CASE ssMethodType OF
    SS_INITIALIZE: 
        temporalCounter_i1(timerAction := 1, maxTime := 0);
        temporalCounter_i2(timerAction := 1, maxTime := 0);
        temporalCounter_i1(timerAction := 1, maxTime := 0);
        is_active_c6_ChiefMaster := 0;
        is_c6_ChiefMaster := ChiefMaster_IN_NO_ACTIVE_CHILD_k;
        REQ_HV_ON := 0.0;
        ContactorState := 0.0;
    SS_OUTPUT: 
        (* Chart: '<S33>/Chart_REQ_HV_ON_Batt3' *)
        (* Gateway: ChiefMaster/Flow Logic/Battery HVControl/REQ_HV_ON_Batt/Chart_REQ_HV_ON_Batt3 *)
        (* During: ChiefMaster/Flow Logic/Battery HVControl/REQ_HV_ON_Batt/Chart_REQ_HV_ON_Batt3 *)

        IF is_active_c6_ChiefMaster = 0 THEN 
            (* Entry: ChiefMaster/Flow Logic/Battery HVControl/REQ_HV_ON_Batt/Chart_REQ_HV_ON_Batt3 *)
            is_active_c6_ChiefMaster := 1;
            (* Entry Internal: ChiefMaster/Flow Logic/Battery HVControl/REQ_HV_ON_Batt/Chart_REQ_HV_ON_Batt3 *)
            (* Transition: '<S42>:8' *)
            is_c6_ChiefMaster := ChiefMaster_IN_Default_f;
            (* Entry 'Default': '<S42>:7' *)
            (* '<S42>:7:2' REQ_HV_ON = 0 *)
            REQ_HV_ON := 0.0;
            (* '<S42>:7:3' ContactorState = 1 *)
            ContactorState := 1.0;
        ELSE 
            temp2 := FALSE;
            temp3 := FALSE;
            temp4 := FALSE;
            temp5 := FALSE;

            CASE is_c6_ChiefMaster OF
                ChiefMaster_IN_CONTACTOR_OFF_f: 
                    (* During 'CONTACTOR_OFF': '<S42>:18' *)
                    (* '<S42>:23:1' sf_internal_predicateOutput = InsulationReadyOK == false ||... *)
                    (* '<S42>:23:2' SDError_BB == true ||... *)
                    (* '<S42>:23:3' Software_Reset_KL15_BB == true ||... *)
                    (* '<S42>:23:4' KL15_CM_disable == true; *)

                    IF ((( NOT InsulationReadyOK) OR SDError_BB) OR (Software_Reset_KL15_BB = 1.0)) OR KL15_CM_disable THEN 
                        (* Transition: '<S42>:23' *)
                        is_c6_ChiefMaster := ChiefMaster_IN_Default_f;
                        (* Entry 'Default': '<S42>:7' *)
                        (* '<S42>:7:2' REQ_HV_ON = 0 *)
                        REQ_HV_ON := 0.0;
                        (* '<S42>:7:3' ContactorState = 1 *)
                        ContactorState := 1.0;
                    ELSE 
                        (* '<S42>:21:1' sf_internal_predicateOutput = after(2,sec) &&... *)
                        (* '<S42>:21:2' IMD_Active_BB1 == false &&... *)
                        (* '<S42>:21:3' IMD_Active_BB2 == false &&... *)
                        (* '<S42>:21:4' IMD_Active_BB3 == true &&... *)
                        (* '<S42>:21:5' MainHV_PlusMinus_Status == 0; *)
                        temporalCounter_i1(timerAction := 2, maxTime := 2000);

                        IF temporalCounter_i1.done THEN 

                            IF ((( NOT IMD_Active_BB1) AND ( NOT IMD_Active_BB2)) AND IMD_Active_BB3) AND ( NOT MainHV_PlusMinus_Status) THEN 
                                (* Transition: '<S42>:21' *)
                                temp3 := TRUE;
                            ELSE 
                                temp5 := TRUE;
                            END_IF;

                        ELSE 
                            temp5 := TRUE;
                        END_IF;

                    END_IF;

                ChiefMaster_IN_CONTACTOR_ON_b: 
                    (* During 'CONTACTOR_ON': '<S42>:20' *)
                    (* '<S42>:44:1' sf_internal_predicateOutput = (KL15_CM_disable == true || SDError_BB == true || System_SD == true) &&... *)
                    (* '<S42>:44:2' (MainHV_SD_OK == true || HV_REL_ON_BB3 == false); *)
                    tmp :=  NOT HV_REL_ON_BB3;

                    IF ((KL15_CM_disable OR SDError_BB) OR System_SD) AND (MainHV_SD_OK OR tmp) THEN 
                        (* Transition: '<S42>:44' *)
                        is_c6_ChiefMaster := ChiefMaster_IN_hold_k;
                        temporalCounter_i1(timerAction := 1, maxTime := 0);
                    ELSE 
                        (* '<S42>:51:1' sf_internal_predicateOutput = SDError_BB == true &&... *)
                        (* '<S42>:51:2' (HV_REL_ON_BB1 == true || HV_REL_ON_BB2 == true) &&... *)
                        (* '<S42>:51:3' (SafeToSD == true || HV_REL_ON_BB3 == false); *)
                        temp1 := HV_REL_ON_BB1 OR HV_REL_ON_BB2;

                        IF (SDError_BB AND temp1) AND (SafeToSD OR tmp) THEN 
                            (* Transition: '<S42>:51' *)
                            temp4 := TRUE;
                        ELSE 
                            (* '<S42>:66:1' sf_internal_predicateOutput = (HV_REL_ON_BB1 == true || HV_REL_ON_BB2 == true) &&... *)
                            (* '<S42>:66:2' REQ_HV_Open == true; *)

                            IF temp1 AND REQ_HV_Open THEN 
                                (* Transition: '<S42>:66' *)
                                temp4 := TRUE;
                            ELSE 
                                (* '<S42>:20:2' REQ_HV_ON = 1 *)
                                REQ_HV_ON := 1.0;
                                (* '<S42>:20:3' ContactorState = 3 *)
                                ContactorState := 3.0;
                            END_IF;

                        END_IF;

                    END_IF;

                ChiefMaster_IN_Default_f: 
                    (* During 'Default': '<S42>:7' *)
                    (* '<S42>:19:1' sf_internal_predicateOutput = IP_boChargeStop_Pressed == false &&... *)
                    (* '<S42>:19:2' KL15_CM_disable == false &&... *)
                    (* '<S42>:19:3' InsulationReadyOK == true &&... *)
                    (* '<S42>:19:4' SDError_BB == false &&... *)
                    (* '<S42>:19:5' System_SD == false; *)

                    IF (((( NOT IP_boChargeStop_Pressed) AND ( NOT KL15_CM_disable)) AND InsulationReadyOK) AND ( NOT SDError_BB)) AND ( NOT System_SD) THEN 
                        (* Transition: '<S42>:19' *)
                        is_c6_ChiefMaster := ChiefMaster_IN_CONTACTOR_OFF_f;
                        temporalCounter_i1(timerAction := 1, maxTime := 0);
                        temporalCounter_i2(timerAction := 1, maxTime := 0);
                        (* Entry 'CONTACTOR_OFF': '<S42>:18' *)
                        (* '<S42>:18:2' REQ_HV_ON = 0 *)
                        REQ_HV_ON := 0.0;
                        (* '<S42>:18:3' ContactorState = 2 *)
                        ContactorState := 2.0;
                    ELSE 
                        (* '<S42>:7:2' REQ_HV_ON = 0 *)
                        REQ_HV_ON := 0.0;
                        (* '<S42>:7:3' ContactorState = 1 *)
                        ContactorState := 1.0;
                    END_IF;

                ELSE
                    (* During 'hold': '<S42>:63' *)
                    (* '<S42>:64:1' sf_internal_predicateOutput = after(2,sec); *)
                    temporalCounter_i1(timerAction := 2, maxTime := 2000);

                    IF temporalCounter_i1.done THEN 
                        (* Transition: '<S42>:64' *)
                        is_c6_ChiefMaster := ChiefMaster_IN_Default_f;
                        (* Entry 'Default': '<S42>:7' *)
                        (* '<S42>:7:2' REQ_HV_ON = 0 *)
                        REQ_HV_ON := 0.0;
                        (* '<S42>:7:3' ContactorState = 1 *)
                        ContactorState := 1.0;
                    END_IF;

            END_CASE;


            IF temp5 THEN 
                (* '<S42>:28:1' sf_internal_predicateOutput = after(2,sec) &&... *)
                (* '<S42>:28:2' IMD_Active_BB3 == false &&... *)
                (* '<S42>:28:3' MainHV_PlusMinus_Status == 1 &&... *)
                (* '<S42>:28:4' (IMD_Active_BB1 == true || IMD_Active_BB2 ==true || IsolationMeasurementRequest == false) &&... *)
                (* '<S42>:28:5' SafeToCloseHV == true; *)
                temporalCounter_i2(timerAction := 2, maxTime := 2000);

                IF temporalCounter_i2.done THEN 

                    IF ((( NOT IMD_Active_BB3) AND MainHV_PlusMinus_Status) AND ((IMD_Active_BB1 OR IMD_Active_BB2) OR ( NOT IsolationMeasurementRequest))) AND SafeToCloseHV_n THEN 
                        (* Transition: '<S42>:28' *)
                        temp3 := TRUE;
                    ELSE 
                        temp2 := TRUE;
                    END_IF;

                ELSE 
                    temp2 := TRUE;
                END_IF;

            END_IF;


            IF temp4 THEN 
                is_c6_ChiefMaster := ChiefMaster_IN_Default_f;
                (* Entry 'Default': '<S42>:7' *)
                (* '<S42>:7:2' REQ_HV_ON = 0 *)
                REQ_HV_ON := 0.0;
                (* '<S42>:7:3' ContactorState = 1 *)
                ContactorState := 1.0;
            END_IF;


            IF temp3 THEN 
                is_c6_ChiefMaster := ChiefMaster_IN_CONTACTOR_ON_b;
                (* Entry 'CONTACTOR_ON': '<S42>:20' *)
                (* '<S42>:20:2' REQ_HV_ON = 1 *)
                REQ_HV_ON := 1.0;
                (* '<S42>:20:3' ContactorState = 3 *)
                ContactorState := 3.0;
            END_IF;


            IF temp2 THEN 
                (* '<S42>:18:2' REQ_HV_ON = 0 *)
                REQ_HV_ON := 0.0;
                (* '<S42>:18:3' ContactorState = 2 *)
                ContactorState := 2.0;
            END_IF;

        END_IF;

        (* End of Chart: '<S33>/Chart_REQ_HV_ON_Batt3' *)
END_CASE;

END_FUNCTION_BLOCK

// Device/Application/Chart_ContactorFB_State_Batt3
FUNCTION_BLOCK Chart_ContactorFB_State_Batt3
VAR_INPUT
	ssMethodType: SINT;
	HV_Minus_Sense_BB: BOOL;
	HV_Plus_Sense_BB: BOOL;
	REQ_HV_ON: LREAL;
END_VAR
VAR_OUTPUT
	Contactor_FB_State: LREAL;
END_VAR
VAR
	temporalCounter_i1: PLC_CODER_TIMER;
	is_c38_ChiefMaster: USINT;
	is_active_c38_ChiefMaster: USINT;
END_VAR



CASE ssMethodType OF
    SS_INITIALIZE: 
        temporalCounter_i1(timerAction := 1, maxTime := 0);
        is_active_c38_ChiefMaster := 0;
        is_c38_ChiefMaster := ChiefMaster_IN_NO_ACTIVE_CHILD_i;
        Contactor_FB_State := 0.0;
    SS_OUTPUT: 
        (* Chart: '<S33>/Chart_ContactorFB_State_Batt3' *)
        (* Gateway: ChiefMaster/Flow Logic/Battery HVControl/REQ_HV_ON_Batt/Chart_ContactorFB_State_Batt3 *)
        (* During: ChiefMaster/Flow Logic/Battery HVControl/REQ_HV_ON_Batt/Chart_ContactorFB_State_Batt3 *)

        IF is_active_c38_ChiefMaster = 0 THEN 
            (* Entry: ChiefMaster/Flow Logic/Battery HVControl/REQ_HV_ON_Batt/Chart_ContactorFB_State_Batt3 *)
            is_active_c38_ChiefMaster := 1;
            (* Entry Internal: ChiefMaster/Flow Logic/Battery HVControl/REQ_HV_ON_Batt/Chart_ContactorFB_State_Batt3 *)
            (* Transition: '<S39>:2' *)
            is_c38_ChiefMaster := ChiefMaster_IN_default_n;
            (* Entry 'default': '<S39>:1' *)
            (* '<S39>:1:2' Contactor_FB_State = 0 *)
            Contactor_FB_State := 0.0;
        ELSE 

            CASE is_c38_ChiefMaster OF
                ChiefMaster_IN_Error_c: 
                    (* During 'Error': '<S39>:12' *)
                    (* '<S39>:51:1' sf_internal_predicateOutput = REQ_HV_ON == 1; *)

                    IF REQ_HV_ON = 1.0 THEN 
                        (* Transition: '<S39>:51' *)
                        is_c38_ChiefMaster := ChiefMaster_IN_default_n;
                        (* Entry 'default': '<S39>:1' *)
                        (* '<S39>:1:2' Contactor_FB_State = 0 *)
                        Contactor_FB_State := 0.0;
                    ELSE 
                        (* '<S39>:12:2' Contactor_FB_State = 3 *)
                        Contactor_FB_State := 3.0;
                    END_IF;

                ChiefMaster_IN_Open_n: 
                    (* During 'Open': '<S39>:46' *)
                    (* '<S39>:50:1' sf_internal_predicateOutput = REQ_HV_ON == 1; *)

                    IF REQ_HV_ON = 1.0 THEN 
                        (* Transition: '<S39>:50' *)
                        is_c38_ChiefMaster := ChiefMaster_IN_default_n;
                        (* Entry 'default': '<S39>:1' *)
                        (* '<S39>:1:2' Contactor_FB_State = 0 *)
                        Contactor_FB_State := 0.0;
                    ELSE 
                        (* '<S39>:46:2' Contactor_FB_State = 1 *)
                        Contactor_FB_State := 1.0;
                    END_IF;

                ChiefMaster_IN_default_n: 
                    (* During 'default': '<S39>:1' *)
                    (* '<S39>:5:1' sf_internal_predicateOutput = REQ_HV_ON == 0; *)

                    IF REQ_HV_ON = 0.0 THEN 
                        (* Transition: '<S39>:5' *)
                        is_c38_ChiefMaster := ChiefMaster_IN_hold_h;
                        temporalCounter_i1(timerAction := 1, maxTime := 0);
                        (* Entry 'hold': '<S39>:4' *)
                        (* '<S39>:4:2' Contactor_FB_State = 0 *)
                        Contactor_FB_State := 0.0;
                    ELSE 
                        (* '<S39>:1:2' Contactor_FB_State = 0 *)
                        Contactor_FB_State := 0.0;
                    END_IF;

                ELSE
                    (* During 'hold': '<S39>:4' *)
                    (* '<S39>:13:1' sf_internal_predicateOutput = after(5,sec); *)
                    temporalCounter_i1(timerAction := 2, maxTime := 5000);

                    IF temporalCounter_i1.done THEN 
                        (* Transition: '<S39>:13' *)
                        is_c38_ChiefMaster := ChiefMaster_IN_Error_c;
                        (* Entry 'Error': '<S39>:12' *)
                        (* '<S39>:12:2' Contactor_FB_State = 3 *)
                        Contactor_FB_State := 3.0;
                    ELSE 
                        (* '<S39>:47:1' sf_internal_predicateOutput = HV_Plus_Sense_BB == false &&... *)
                        (* '<S39>:47:2' HV_Minus_Sense_BB == false; *)

                        IF ( NOT HV_Plus_Sense_BB) AND ( NOT HV_Minus_Sense_BB) THEN 
                            (* Transition: '<S39>:47' *)
                            is_c38_ChiefMaster := ChiefMaster_IN_Open_n;
                            (* Entry 'Open': '<S39>:46' *)
                            (* '<S39>:46:2' Contactor_FB_State = 1 *)
                            Contactor_FB_State := 1.0;
                        ELSE 
                            (* '<S39>:4:2' Contactor_FB_State = 0 *)
                            Contactor_FB_State := 0.0;
                        END_IF;

                    END_IF;

            END_CASE;

        END_IF;

        (* End of Chart: '<S33>/Chart_ContactorFB_State_Batt3' *)
END_CASE;

END_FUNCTION_BLOCK

// Device/Application/Chart_PrechargeStatus
FUNCTION_BLOCK Chart_PrechargeStatus
VAR_INPUT
	ssMethodType: SINT;
	REQ_MainHV_ON_Precharge: BOOL;
	LoadCurrent: BOOL;
	LoadVoltage: REAL;
	SystemVoltage: REAL;
	KL15_CM_diable: BOOL;
	MainHV_Minus_Status: LREAL;
END_VAR
VAR_OUTPUT
	Precharge_Satus: LREAL;
END_VAR
VAR
	temporalCounter_i2: PLC_CODER_TIMER;
	temporalCounter_i1: PLC_CODER_TIMER;
	is_c21_ChiefMaster: USINT;
	is_active_c21_ChiefMaster: USINT;
	temp1: BOOL;
END_VAR



CASE ssMethodType OF
    SS_INITIALIZE: 
        temporalCounter_i1(timerAction := 1, maxTime := 0);
        temporalCounter_i2(timerAction := 1, maxTime := 0);
        is_active_c21_ChiefMaster := 0;
        is_c21_ChiefMaster := ChiefMaster_IN_NO_ACTIVE_CHILD;
        Precharge_Satus := 0.0;
    SS_OUTPUT: 
        (* Chart: '<S13>/Chart_PrechargeStatus' *)
        (* Gateway: ChiefMaster/Flow Logic/BDU Control/BDUSystem/Chart_PrechargeStatus *)
        (* During: ChiefMaster/Flow Logic/BDU Control/BDUSystem/Chart_PrechargeStatus *)

        IF is_active_c21_ChiefMaster = 0 THEN 
            (* Entry: ChiefMaster/Flow Logic/BDU Control/BDUSystem/Chart_PrechargeStatus *)
            is_active_c21_ChiefMaster := 1;
            (* Entry Internal: ChiefMaster/Flow Logic/BDU Control/BDUSystem/Chart_PrechargeStatus *)
            (* Transition: '<S15>:4' *)
            is_c21_ChiefMaster := ChiefMaster_IN_Default;
            (* Entry 'Default': '<S15>:3' *)
            (* '<S15>:3:2' Precharge_Satus = 0 *)
            Precharge_Satus := 0.0;
        ELSE 

            CASE is_c21_ChiefMaster OF
                ChiefMaster_IN_Default: 
                    (* During 'Default': '<S15>:3' *)
                    (* '<S15>:20:1' sf_internal_predicateOutput = REQ_MainHV_ON_Precharge == true &&... *)
                    (* '<S15>:20:2' KL15_CM_diable == false; *)

                    IF REQ_MainHV_ON_Precharge AND ( NOT KL15_CM_diable) THEN 
                        (* Transition: '<S15>:20' *)
                        is_c21_ChiefMaster := ChiefMaster_IN_delay1;
                        temporalCounter_i1(timerAction := 1, maxTime := 0);
                        temporalCounter_i2(timerAction := 1, maxTime := 0);
                    ELSE 
                        (* '<S15>:3:2' Precharge_Satus = 0 *)
                        Precharge_Satus := 0.0;
                    END_IF;

                ChiefMaster_IN_PrechargeFail: 
                    (* During 'PrechargeFail': '<S15>:28' *)
                    (* Transition: '<S15>:37' *)
                    (* Transition: '<S15>:38' *)
                    (* '<S15>:35:1' sf_internal_predicateOutput = KL15_CM_diable == true; *)

                    IF KL15_CM_diable THEN 
                        (* Transition: '<S15>:35' *)
                        is_c21_ChiefMaster := ChiefMaster_IN_Default;
                        (* Entry 'Default': '<S15>:3' *)
                        (* '<S15>:3:2' Precharge_Satus = 0 *)
                        Precharge_Satus := 0.0;
                    ELSE 
                        (* '<S15>:28:2' Precharge_Satus = 2 *)
                        Precharge_Satus := 2.0;
                    END_IF;

                ChiefMaster_IN_PrechargeSuccess: 
                    (* During 'PrechargeSuccess': '<S15>:19' *)
                    (* Transition: '<S15>:32' *)
                    (* Transition: '<S15>:45' *)
                    (* '<S15>:46:1' sf_internal_predicateOutput = MainHV_Minus_Status == 1 ||... *)
                    (* '<S15>:46:2' MainHV_Minus_Status == 3; *)

                    IF (MainHV_Minus_Status = 1.0) OR (MainHV_Minus_Status = 3.0) THEN 
                        (* Transition: '<S15>:46' *)
                        is_c21_ChiefMaster := ChiefMaster_IN_Default;
                        (* Entry 'Default': '<S15>:3' *)
                        (* '<S15>:3:2' Precharge_Satus = 0 *)
                        Precharge_Satus := 0.0;
                    ELSE 
                        (* '<S15>:19:2' Precharge_Satus = 1 *)
                        Precharge_Satus := 1.0;
                    END_IF;

                ELSE
                    (* During 'delay1': '<S15>:26' *)
                    (* '<S15>:27:1' sf_internal_predicateOutput = after(500,msec) &&... *)
                    (* '<S15>:27:2' LoadCurrent == 0 &&... *)
                    (* '<S15>:27:3' abs(LoadVoltage - SystemVoltage) <= 5; *)
                    temp1 := FALSE;
                    temporalCounter_i2(timerAction := 2, maxTime := 500);

                    IF temporalCounter_i2.done THEN 

                        IF  NOT LoadCurrent THEN 

                            IF ABS(LoadVoltage - SystemVoltage) <= 5.0 THEN 
                                (* Transition: '<S15>:27' *)
                                is_c21_ChiefMaster := ChiefMaster_IN_PrechargeSuccess;
                                (* Entry 'PrechargeSuccess': '<S15>:19' *)
                                (* '<S15>:19:2' Precharge_Satus = 1 *)
                                Precharge_Satus := 1.0;
                            ELSE 
                                temp1 := TRUE;
                            END_IF;

                        ELSE 
                            temp1 := TRUE;
                        END_IF;

                    ELSE 
                        temp1 := TRUE;
                    END_IF;

                    temporalCounter_i1(timerAction := 2, maxTime := 3000);

                    IF temp1 AND temporalCounter_i1.done THEN 
                        (* '<S15>:25:1' sf_internal_predicateOutput = after(3,sec); *)
                        (* Transition: '<S15>:25' *)
                        is_c21_ChiefMaster := ChiefMaster_IN_PrechargeFail;
                        (* Entry 'PrechargeFail': '<S15>:28' *)
                        (* '<S15>:28:2' Precharge_Satus = 2 *)
                        Precharge_Satus := 2.0;
                    END_IF;

            END_CASE;

        END_IF;

        (* End of Chart: '<S13>/Chart_PrechargeStatus' *)
END_CASE;

END_FUNCTION_BLOCK

// Device/Application/Chart_SetDominantSwitch
FUNCTION_BLOCK Chart_SetDominantSwitch
VAR_INPUT
	ssMethodType: SINT;
	boData_In: BOOL;
	boReset: BOOL;
END_VAR
VAR_OUTPUT
	boData_Out: BOOL;
END_VAR
VAR
	is_active_c3_Library_DataProcessing_v1_1: USINT;
	is_c3_Library_DataProcessing_v1_1: USINT;
END_VAR



CASE ssMethodType OF
    SS_INITIALIZE: 
        is_active_c3_Library_DataProcessing_v1_1 := 0;
        is_c3_Library_DataProcessing_v1_1 := ChiefMaster_IN_NO_ACTIVE_CHILD_cn;
        boData_Out := FALSE;
    SS_OUTPUT: 
        (* Chart: '<S149>/Chart_SetDominantSwitch' *)
        (* Gateway: Lib_SetDominantSwitch/Chart_SetDominantSwitch *)
        (* During: Lib_SetDominantSwitch/Chart_SetDominantSwitch *)

        IF is_active_c3_Library_DataProcessing_v1_1 = 0 THEN 
            (* Entry: Lib_SetDominantSwitch/Chart_SetDominantSwitch *)
            is_active_c3_Library_DataProcessing_v1_1 := 1;
            (* Entry Internal: Lib_SetDominantSwitch/Chart_SetDominantSwitch *)
            (* Transition: '<S152>:10' *)
            is_c3_Library_DataProcessing_v1_1 := ChiefMaster_IN_Initial_state_g;
            (* Entry 'Initial_state': '<S152>:12' *)
            (* '<S152>:12:3' boData_Out = false; *)
            boData_Out := FALSE;
        ELSE 

            CASE is_c3_Library_DataProcessing_v1_1 OF
                ChiefMaster_IN_Initial_state_g: 
                    (* During 'Initial_state': '<S152>:12' *)
                    (* '<S152>:9:1' sf_internal_predicateOutput = boData_In == true; *)

                    IF boData_In THEN 
                        (* Transition: '<S152>:9' *)
                        is_c3_Library_DataProcessing_v1_1 := ChiefMaster_IN_state1_o;
                        (* Entry 'state1': '<S152>:6' *)
                        (* '<S152>:6:3' boData_Out = true; *)
                        boData_Out := TRUE;
                    ELSE 
                        (* '<S152>:12:3' boData_Out = false; *)
                        boData_Out := FALSE;
                    END_IF;

                ChiefMaster_IN_Reset_state_b: 
                    (* During 'Reset_state': '<S152>:4' *)
                    (* '<S152>:5:1' sf_internal_predicateOutput = boReset == false; *)

                    IF  NOT boReset THEN 
                        (* Transition: '<S152>:5' *)
                        is_c3_Library_DataProcessing_v1_1 := ChiefMaster_IN_Initial_state_g;
                        (* Entry 'Initial_state': '<S152>:12' *)
                        (* '<S152>:12:3' boData_Out = false; *)
                        boData_Out := FALSE;
                    ELSE 
                        (* '<S152>:4:3' boData_Out = false; *)
                        boData_Out := FALSE;
                    END_IF;

                ChiefMaster_IN_state1_o: 
                    (* During 'state1': '<S152>:6' *)
                    (* '<S152>:7:1' sf_internal_predicateOutput = boData_In == false; *)

                    IF  NOT boData_In THEN 
                        (* Transition: '<S152>:7' *)
                        is_c3_Library_DataProcessing_v1_1 := ChiefMaster_IN_state2_e;
                        (* Entry 'state2': '<S152>:8' *)
                        (* '<S152>:8:3' boData_Out = true; *)
                        boData_Out := TRUE;
                    ELSE 
                        (* '<S152>:6:3' boData_Out = true; *)
                        boData_Out := TRUE;
                    END_IF;

                ELSE
                    (* During 'state2': '<S152>:8' *)
                    (* '<S152>:11:1' sf_internal_predicateOutput = boReset == true; *)

                    IF boReset THEN 
                        (* Transition: '<S152>:11' *)
                        is_c3_Library_DataProcessing_v1_1 := ChiefMaster_IN_Reset_state_b;
                        (* Entry 'Reset_state': '<S152>:4' *)
                        (* '<S152>:4:3' boData_Out = false; *)
                        boData_Out := FALSE;
                    ELSE 
                        (* '<S152>:8:3' boData_Out = true; *)
                        boData_Out := TRUE;
                    END_IF;

            END_CASE;

        END_IF;

        (* End of Chart: '<S149>/Chart_SetDominantSwitch' *)
END_CASE;

END_FUNCTION_BLOCK

// Device/Application/EmergencySD
FUNCTION_BLOCK EmergencySD
VAR_INPUT
	ssMethodType: SINT;
	FL_boKL15_Reset: BOOL;
	IT_boEmergencySwitch_NC: BOOL;
	IT_boEmergencySwitch_NO: BOOL;
	IT_boHW_HVIL_BDU: BOOL;
	IT_boHW_HVIL_Components: BOOL;
	IT_boHW_HVIL_Battery: BOOL;
	IT_boHW_HVIL_Overrule: BOOL;
	IT_boHW_ResetButton_LED_NO_State: BOOL;
END_VAR
VAR_OUTPUT
	FL_boSS_System_ESD: BOOL;
	FL_u8SS_EmergencyStopState: USINT;
	FL_boHVIL_NOK: BOOL;
END_VAR
VAR
	is_active_c55_ChiefMaster: USINT;
	is_c55_ChiefMaster: USINT;
	temporalCounter_i1: PLC_CODER_TIMER;
	is_active_c28_ChiefMaster: USINT;
	is_c28_ChiefMaster: USINT;
	temporalCounter_i1_h: PLC_CODER_TIMER;
	i0_fcn_EmergencyButtonState: fcn_EmergencyButtonState;
	i0_HVIL_NOK: HVIL_NOK;
	rtb_out_j1: BOOL;
	rtb_out_h: BOOL;
	rtb_TmpSignalConversionAtfcn_EmergencyButtonStateInport2: BOOL;
END_VAR



CASE ssMethodType OF
    SS_INITIALIZE: 
        (* SystemInitialize for Chart: '<S140>/EmergencySwitch_Input_Delay1' *)
        temporalCounter_i1(timerAction := 1, maxTime := 0);
        is_active_c55_ChiefMaster := 0;
        is_c55_ChiefMaster := ChiefMaster_IN_NO_ACTIVE_CHILD_l;
        (* SystemInitialize for Chart: '<S140>/EmergencySwitch_Input_Delay' *)
        temporalCounter_i1_h(timerAction := 1, maxTime := 0);
        is_active_c28_ChiefMaster := 0;
        is_c28_ChiefMaster := ChiefMaster_IN_NO_ACTIVE_CHILD_l;
        (* SystemInitialize for Chart: '<S140>/EmergencySwitch_Input_Delay1' incorporates:
         *  Chart: '<S140>/EmergencySwitch_Input_Delay' *)
        i0_fcn_EmergencyButtonState(ssMethodType := SS_INITIALIZE, IP_boVS_EmergencySwitch_NO_S1 := FALSE, IP_boVS_EmergencySwitch_NC_S2 := rtb_TmpSignalConversionAtfcn_EmergencyButtonStateInport2, IP_boVS_EmergencySwitch_NC_S3 := FALSE, b_reset := rtb_TmpSignalConversionAtfcn_EmergencyButtonStateInport2);
        FL_u8SS_EmergencyStopState := i0_fcn_EmergencyButtonState.FL_u8VS_EmergencyStopState;
        i0_HVIL_NOK(ssMethodType := SS_INITIALIZE, boReset := rtb_TmpSignalConversionAtfcn_EmergencyButtonStateInport2, IT_boHW_HVIL_BDU := IT_boHW_HVIL_BDU, IT_boHW_HVIL_Components := IT_boHW_HVIL_Components, IT_boHW_HVIL_Battery := IT_boHW_HVIL_Battery);
    SS_OUTPUT: 
        (* Logic: '<S112>/AND' incorporates:
         *  Logic: '<S112>/NOT' *)
        rtb_TmpSignalConversionAtfcn_EmergencyButtonStateInport2 := IT_boHW_ResetButton_LED_NO_State AND ( NOT FL_boKL15_Reset);
        (* Chart: '<S140>/EmergencySwitch_Input_Delay1' *)
        (* Gateway: ChiefMaster/Flow Logic/System Status/EmergencySD/Emergency_Switch_Control/EmergencySwitch_Input_Delay1 *)
        (* During: ChiefMaster/Flow Logic/System Status/EmergencySD/Emergency_Switch_Control/EmergencySwitch_Input_Delay1 *)

        IF is_active_c55_ChiefMaster = 0 THEN 
            (* Entry: ChiefMaster/Flow Logic/System Status/EmergencySD/Emergency_Switch_Control/EmergencySwitch_Input_Delay1 *)
            is_active_c55_ChiefMaster := 1;
            (* Entry Internal: ChiefMaster/Flow Logic/System Status/EmergencySD/Emergency_Switch_Control/EmergencySwitch_Input_Delay1 *)
            (* Transition: '<S143>:2' *)
            is_c55_ChiefMaster := ChiefMaster_IN_Initial;
            (* Entry 'Initial': '<S143>:1' *)
            (* '<S143>:1:3' out = IP_boVS_EmergensySwitch; *)
            rtb_out_j1 := IT_boEmergencySwitch_NO;
        ELSE 

            CASE is_c55_ChiefMaster OF
                ChiefMaster_IN_After_delay: 
                    (* During 'After_delay': '<S143>:4' *)
                    (* '<S143>:10:1' sf_internal_predicateOutput = IP_boVS_EmergensySwitch == true; *)

                    IF IT_boEmergencySwitch_NO THEN 
                        (* Transition: '<S143>:10' *)
                        is_c55_ChiefMaster := ChiefMaster_IN_Initial;
                        (* Entry 'Initial': '<S143>:1' *)
                        (* '<S143>:1:3' out = IP_boVS_EmergensySwitch; *)
                        rtb_out_j1 := TRUE;
                    ELSE 
                        (* '<S143>:4:3' out = IP_boVS_EmergensySwitch; *)
                        rtb_out_j1 := FALSE;
                    END_IF;

                ChiefMaster_IN_Delay_a: 
                    (* During 'Delay': '<S143>:3' *)
                    (* '<S143>:6:1' sf_internal_predicateOutput = after(10, msec); *)
                    temporalCounter_i1(timerAction := 2, maxTime := 10);

                    IF temporalCounter_i1.done THEN 
                        (* Transition: '<S143>:6' *)
                        is_c55_ChiefMaster := ChiefMaster_IN_After_delay;
                        (* Entry 'After_delay': '<S143>:4' *)
                        (* '<S143>:4:3' out = IP_boVS_EmergensySwitch; *)
                        rtb_out_j1 := IT_boEmergencySwitch_NO;
                    ELSE 
                        (* '<S143>:3:3' out = false; *)
                        rtb_out_j1 := FALSE;
                    END_IF;

                ELSE
                    (* During 'Initial': '<S143>:1' *)
                    (* '<S143>:5:1' sf_internal_predicateOutput = IP_boVS_EmergensySwitch == false; *)

                    IF  NOT IT_boEmergencySwitch_NO THEN 
                        (* Transition: '<S143>:5' *)
                        is_c55_ChiefMaster := ChiefMaster_IN_Delay_a;
                        temporalCounter_i1(timerAction := 1, maxTime := 0);
                        (* Entry 'Delay': '<S143>:3' *)
                        (* '<S143>:3:3' out = false; *)
                        rtb_out_j1 := FALSE;
                    ELSE 
                        (* '<S143>:1:3' out = IP_boVS_EmergensySwitch; *)
                        rtb_out_j1 := TRUE;
                    END_IF;

            END_CASE;

        END_IF;

        (* End of Chart: '<S140>/EmergencySwitch_Input_Delay1' *)
        

        (* Chart: '<S140>/EmergencySwitch_Input_Delay' *)
        (* Gateway: ChiefMaster/Flow Logic/System Status/EmergencySD/Emergency_Switch_Control/EmergencySwitch_Input_Delay *)
        (* During: ChiefMaster/Flow Logic/System Status/EmergencySD/Emergency_Switch_Control/EmergencySwitch_Input_Delay *)

        IF is_active_c28_ChiefMaster = 0 THEN 
            (* Entry: ChiefMaster/Flow Logic/System Status/EmergencySD/Emergency_Switch_Control/EmergencySwitch_Input_Delay *)
            is_active_c28_ChiefMaster := 1;
            (* Entry Internal: ChiefMaster/Flow Logic/System Status/EmergencySD/Emergency_Switch_Control/EmergencySwitch_Input_Delay *)
            (* Transition: '<S142>:2' *)
            is_c28_ChiefMaster := ChiefMaster_IN_Initial;
            (* Entry 'Initial': '<S142>:1' *)
            (* '<S142>:1:3' out = IP_boVS_EmergensySwitch; *)
            rtb_out_h := IT_boEmergencySwitch_NC;
        ELSE 

            CASE is_c28_ChiefMaster OF
                ChiefMaster_IN_After_delay: 
                    (* During 'After_delay': '<S142>:4' *)
                    (* '<S142>:10:1' sf_internal_predicateOutput = IP_boVS_EmergensySwitch == true; *)

                    IF IT_boEmergencySwitch_NC THEN 
                        (* Transition: '<S142>:10' *)
                        is_c28_ChiefMaster := ChiefMaster_IN_Initial;
                        (* Entry 'Initial': '<S142>:1' *)
                        (* '<S142>:1:3' out = IP_boVS_EmergensySwitch; *)
                        rtb_out_h := TRUE;
                    ELSE 
                        (* '<S142>:4:3' out = IP_boVS_EmergensySwitch; *)
                        rtb_out_h := FALSE;
                    END_IF;

                ChiefMaster_IN_Delay_a: 
                    (* During 'Delay': '<S142>:3' *)
                    (* '<S142>:6:1' sf_internal_predicateOutput = after(10, msec); *)
                    temporalCounter_i1_h(timerAction := 2, maxTime := 10);

                    IF temporalCounter_i1_h.done THEN 
                        (* Transition: '<S142>:6' *)
                        is_c28_ChiefMaster := ChiefMaster_IN_After_delay;
                        (* Entry 'After_delay': '<S142>:4' *)
                        (* '<S142>:4:3' out = IP_boVS_EmergensySwitch; *)
                        rtb_out_h := IT_boEmergencySwitch_NC;
                    ELSE 
                        (* '<S142>:3:3' out = true; *)
                        rtb_out_h := TRUE;
                    END_IF;

                ELSE
                    (* During 'Initial': '<S142>:1' *)
                    (* '<S142>:5:1' sf_internal_predicateOutput = IP_boVS_EmergensySwitch == false; *)

                    IF  NOT IT_boEmergencySwitch_NC THEN 
                        (* Transition: '<S142>:5' *)
                        is_c28_ChiefMaster := ChiefMaster_IN_Delay_a;
                        temporalCounter_i1_h(timerAction := 1, maxTime := 0);
                        (* Entry 'Delay': '<S142>:3' *)
                        (* '<S142>:3:3' out = true; *)
                        rtb_out_h := TRUE;
                    ELSE 
                        (* '<S142>:1:3' out = IP_boVS_EmergensySwitch; *)
                        rtb_out_h := TRUE;
                    END_IF;

            END_CASE;

        END_IF;

        (* End of Chart: '<S140>/EmergencySwitch_Input_Delay' *)
        

        (* SignalConversion: '<S140>/TmpSignal ConversionAtfcn_EmergencyButtonStateInport2' *)
        i0_fcn_EmergencyButtonState(ssMethodType := SS_OUTPUT, IP_boVS_EmergencySwitch_NO_S1 := rtb_out_j1, IP_boVS_EmergencySwitch_NC_S2 := rtb_out_h, IP_boVS_EmergencySwitch_NC_S3 := rtb_out_h, b_reset := rtb_TmpSignalConversionAtfcn_EmergencyButtonStateInport2);
        FL_u8SS_EmergencyStopState := i0_fcn_EmergencyButtonState.FL_u8VS_EmergencyStopState;
        i0_HVIL_NOK(ssMethodType := SS_OUTPUT, boReset := rtb_TmpSignalConversionAtfcn_EmergencyButtonStateInport2, IT_boHW_HVIL_BDU := IT_boHW_HVIL_BDU, IT_boHW_HVIL_Components := IT_boHW_HVIL_Components, IT_boHW_HVIL_Battery := IT_boHW_HVIL_Battery);
        FL_boSS_System_ESD := i0_HVIL_NOK.FL_boSS_HVIL_NOK;
        (* Switch: '<S112>/Switch' incorporates:
         *  Constant: '<S112>/Constant' *)

        IF IT_boHW_HVIL_Overrule THEN 
            FL_boHVIL_NOK := FALSE;
        ELSE 
            FL_boHVIL_NOK := FL_boSS_System_ESD;
        END_IF;

        (* End of Switch: '<S112>/Switch' *)
        

        (* Logic: '<S112>/OR1' incorporates:
         *  Constant: '<S139>/Constant'
         *  RelationalOperator: '<S139>/Compare' *)
        FL_boSS_System_ESD := (FL_u8SS_EmergencyStopState >= 1) OR FL_boHVIL_NOK;
END_CASE;

END_FUNCTION_BLOCK

// Device/Application/fcn_EmergencyButtonState
FUNCTION_BLOCK fcn_EmergencyButtonState
VAR_INPUT
	ssMethodType: SINT;
	IP_boVS_EmergencySwitch_NO_S1: BOOL;
	IP_boVS_EmergencySwitch_NC_S2: BOOL;
	IP_boVS_EmergencySwitch_NC_S3: BOOL;
	b_reset: BOOL;
END_VAR
VAR_OUTPUT
	FL_u8VS_EmergencyStopState: USINT;
END_VAR
VAR
	is_active_c29_ChiefMaster: USINT;
	is_c29_ChiefMaster: USINT;
	In_prv: USINT;
END_VAR



CASE ssMethodType OF
    SS_INITIALIZE: 
        (* SystemInitialize for Chart: '<S144>/Chart' *)
        is_active_c29_ChiefMaster := 0;
        is_c29_ChiefMaster := ChiefMaster_IN_NO_ACTIVE_CHILD_b;
        In_prv := 0;
        FL_u8VS_EmergencyStopState := 0;
    SS_OUTPUT: 
        (* Switch: '<S144>/Switch1' incorporates:
         *  Constant: '<S144>/NotPressed'
         *  Logic: '<S144>/AND1'
         *  Logic: '<S144>/AND3'
         *  Logic: '<S144>/AND4'
         *  Logic: '<S144>/AND5'
         *  Switch: '<S144>/Switch' *)

        IF ( NOT IP_boVS_EmergencySwitch_NO_S1) AND (IP_boVS_EmergencySwitch_NC_S2 AND IP_boVS_EmergencySwitch_NC_S3) THEN 
            FL_u8VS_EmergencyStopState := 0;
        ELSIF IP_boVS_EmergencySwitch_NO_S1 AND (( NOT IP_boVS_EmergencySwitch_NC_S2) AND ( NOT IP_boVS_EmergencySwitch_NC_S3)) THEN 
            (* Switch: '<S144>/Switch' incorporates:
             *  Constant: '<S144>/Pressed' *)
            FL_u8VS_EmergencyStopState := 1;
        ELSE 
            (* Switch: '<S144>/Switch' incorporates:
             *  Constant: '<S144>/Error' *)
            FL_u8VS_EmergencyStopState := 2;
        END_IF;

        (* End of Switch: '<S144>/Switch1' *)
        

        (* Chart: '<S144>/Chart' *)
        (* Gateway: ChiefMaster/Flow Logic/System Status/EmergencySD/Emergency_Switch_Control/fcn_EmergencyButtonState/Chart *)
        (* During: ChiefMaster/Flow Logic/System Status/EmergencySD/Emergency_Switch_Control/fcn_EmergencyButtonState/Chart *)

        IF is_active_c29_ChiefMaster = 0 THEN 
            (* Entry: ChiefMaster/Flow Logic/System Status/EmergencySD/Emergency_Switch_Control/fcn_EmergencyButtonState/Chart *)
            is_active_c29_ChiefMaster := 1;
            (* Entry Internal: ChiefMaster/Flow Logic/System Status/EmergencySD/Emergency_Switch_Control/fcn_EmergencyButtonState/Chart *)
            (* Transition: '<S145>:5' *)
            is_c29_ChiefMaster := ChiefMaster_IN_Initial_state;
            (* Entry 'Initial_state': '<S145>:7' *)
            (* '<S145>:7:3' Out = In; *)
        ELSE 

            CASE is_c29_ChiefMaster OF
                ChiefMaster_IN_Initial_state: 
                    (* During 'Initial_state': '<S145>:7' *)
                    (* '<S145>:9:1' sf_internal_predicateOutput = In > uint8(0); *)

                    IF FL_u8VS_EmergencyStopState > 0 THEN 
                        (* Transition: '<S145>:9' *)
                        is_c29_ChiefMaster := ChiefMaster_IN_state1;
                        (* Entry 'state1': '<S145>:2' *)
                        (* '<S145>:2:3' Out = In; *)
                        (* '<S145>:2:4' In_prv = In; *)
                        In_prv := FL_u8VS_EmergencyStopState;
                    END_IF;

                ChiefMaster_IN_Reset_state: 
                    (* During 'Reset_state': '<S145>:1' *)
                    (* '<S145>:8:1' sf_internal_predicateOutput = reset == false; *)

                    IF  NOT b_reset THEN 
                        (* Transition: '<S145>:8' *)
                        is_c29_ChiefMaster := ChiefMaster_IN_Initial_state;
                        (* Entry 'Initial_state': '<S145>:7' *)
                        (* '<S145>:7:3' Out = In; *)
                    ELSE 
                        (* '<S145>:1:3' Out = uint8(0); *)
                        FL_u8VS_EmergencyStopState := 0;
                    END_IF;

                ChiefMaster_IN_state1: 
                    (* During 'state1': '<S145>:2' *)
                    (* '<S145>:6:1' sf_internal_predicateOutput = In == uint8(0); *)

                    IF FL_u8VS_EmergencyStopState = 0 THEN 
                        (* Transition: '<S145>:6' *)
                        is_c29_ChiefMaster := ChiefMaster_IN_state2;
                        (* Entry 'state2': '<S145>:3' *)
                        (* '<S145>:3:3' Out = In_prv; *)
                        FL_u8VS_EmergencyStopState := In_prv;
                    ELSE 
                        (* '<S145>:2:3' Out = In; *)
                        (* '<S145>:2:4' In_prv = In; *)
                        In_prv := FL_u8VS_EmergencyStopState;
                    END_IF;

                ELSE
                    (* During 'state2': '<S145>:3' *)
                    (* '<S145>:4:1' sf_internal_predicateOutput = reset == true; *)

                    IF b_reset THEN 
                        (* Transition: '<S145>:4' *)
                        is_c29_ChiefMaster := ChiefMaster_IN_Reset_state;
                        (* Entry 'Reset_state': '<S145>:1' *)
                        (* '<S145>:1:3' Out = uint8(0); *)
                        FL_u8VS_EmergencyStopState := 0;
                    ELSE 
                        (* '<S145>:3:3' Out = In_prv; *)
                        FL_u8VS_EmergencyStopState := In_prv;
                    END_IF;

            END_CASE;

        END_IF;

        (* End of Chart: '<S144>/Chart' *)
END_CASE;

END_FUNCTION_BLOCK

// Device/Application/HVIL_NOK
FUNCTION_BLOCK HVIL_NOK
VAR_INPUT
	ssMethodType: SINT;
	boReset: BOOL;
	IT_boHW_HVIL_BDU: BOOL;
	IT_boHW_HVIL_Components: BOOL;
	IT_boHW_HVIL_Battery: BOOL;
END_VAR
VAR_OUTPUT
	FL_boSS_HVIL_NOK: BOOL;
END_VAR
VAR
	i0_Chart_SetDominantSwitch: Chart_SetDominantSwitch;
	i1_Chart_SetDominantSwitch: Chart_SetDominantSwitch;
	i2_Chart_SetDominantSwitch: Chart_SetDominantSwitch;
	rtb_Compare_jkc: BOOL;
	rtb_boData_Out_f5: BOOL;
	rtb_Compare_h3: BOOL;
	rtb_Compare_n45: BOOL;
END_VAR



CASE ssMethodType OF
    SS_INITIALIZE: 
        i0_Chart_SetDominantSwitch(ssMethodType := SS_INITIALIZE, boData_In := rtb_Compare_jkc, boReset := boReset);
        rtb_boData_Out_f5 := i0_Chart_SetDominantSwitch.boData_Out;
        i1_Chart_SetDominantSwitch(ssMethodType := SS_INITIALIZE, boData_In := rtb_Compare_h3, boReset := boReset);
        rtb_Compare_jkc := i1_Chart_SetDominantSwitch.boData_Out;
        i2_Chart_SetDominantSwitch(ssMethodType := SS_INITIALIZE, boData_In := rtb_Compare_n45, boReset := boReset);
        rtb_Compare_h3 := i2_Chart_SetDominantSwitch.boData_Out;
    SS_OUTPUT: 
        (* RelationalOperator: '<S146>/Compare' *)
        i0_Chart_SetDominantSwitch(ssMethodType := SS_OUTPUT, boData_In :=  NOT IT_boHW_HVIL_BDU, boReset := boReset);
        rtb_boData_Out_f5 := i0_Chart_SetDominantSwitch.boData_Out;
        (* RelationalOperator: '<S147>/Compare' *)
        i1_Chart_SetDominantSwitch(ssMethodType := SS_OUTPUT, boData_In :=  NOT IT_boHW_HVIL_Components, boReset := boReset);
        rtb_Compare_jkc := i1_Chart_SetDominantSwitch.boData_Out;
        (* RelationalOperator: '<S148>/Compare' *)
        i2_Chart_SetDominantSwitch(ssMethodType := SS_OUTPUT, boData_In :=  NOT IT_boHW_HVIL_Battery, boReset := boReset);
        rtb_Compare_h3 := i2_Chart_SetDominantSwitch.boData_Out;
        (* Logic: '<S141>/OR' *)
        FL_boSS_HVIL_NOK := (rtb_boData_Out_f5 OR rtb_Compare_jkc) OR rtb_Compare_h3;
END_CASE;

END_FUNCTION_BLOCK

// Device/Application/Input_Delay
FUNCTION_BLOCK Input_Delay
VAR_INPUT
	ssMethodType: SINT;
	IP_u8HW_IN_delay_ms_m: UINT;
	Input: BOOL;
END_VAR
VAR_OUTPUT
	out: BOOL;
END_VAR
VAR
	is_active_c2_ChiefMaster: USINT;
	is_c2_ChiefMaster: USINT;
	temporalCounter_i1: PLC_CODER_TIMER;
END_VAR



CASE ssMethodType OF
    SS_INITIALIZE: 
        temporalCounter_i1(timerAction := 1, maxTime := 0);
        is_active_c2_ChiefMaster := 0;
        is_c2_ChiefMaster := ChiefMaster_IN_NO_ACTIVE_CHILD_an;
        out := FALSE;
    SS_OUTPUT: 
        (* Chart: '<S392>/Input_Delay' *)
        (* Gateway: ChiefMaster/Input Processing/HW Inputs/Subsystem/Input_Delay *)
        (* During: ChiefMaster/Input Processing/HW Inputs/Subsystem/Input_Delay *)

        IF is_active_c2_ChiefMaster = 0 THEN 
            (* Entry: ChiefMaster/Input Processing/HW Inputs/Subsystem/Input_Delay *)
            is_active_c2_ChiefMaster := 1;
            (* Entry Internal: ChiefMaster/Input Processing/HW Inputs/Subsystem/Input_Delay *)
            (* Transition: '<S418>:2' *)
            is_c2_ChiefMaster := ChiefMaster_IN_Initial_k;
            temporalCounter_i1(timerAction := 1, maxTime := 0);
            (* Entry 'Initial': '<S418>:1' *)
            (* '<S418>:1:3' out = true; *)
            out := TRUE;
        ELSE 

            CASE is_c2_ChiefMaster OF
                ChiefMaster_IN_After_delay_p: 
                    (* During 'After_delay': '<S418>:4' *)
                    (* '<S418>:4:3' out = Input; *)
                    out := Input;
                ELSE
                    (* During 'Initial': '<S418>:1' *)
                    (* '<S418>:6:1' sf_internal_predicateOutput = after(IP_u8HW_IN_delay_ms, msec); *)
                    temporalCounter_i1(timerAction := 2, maxTime := UINT_TO_DINT(IP_u8HW_IN_delay_ms_m));

                    IF temporalCounter_i1.done THEN 
                        (* Transition: '<S418>:6' *)
                        is_c2_ChiefMaster := ChiefMaster_IN_After_delay_p;
                        (* Entry 'After_delay': '<S418>:4' *)
                        (* '<S418>:4:3' out = Input; *)
                        out := Input;
                    ELSE 
                        (* '<S418>:1:3' out = true; *)
                        out := TRUE;
                    END_IF;

            END_CASE;

        END_IF;

        (* End of Chart: '<S392>/Input_Delay' *)
END_CASE;

END_FUNCTION_BLOCK

// Device/Application/SDError
FUNCTION_BLOCK SDError
VAR_INPUT
	ssMethodType: SINT;
	FL_boKL15_Reset: BOOL;
	IT_Databus: USINT;
	IT_Databus_m: BOOL;
	IT_Databus_n: BOOL;
	IT_Databus_a: BOOL;
	IT_Databus_o: BOOL;
	IT_Databus_or: BOOL;
	IT_Databus_i: BOOL;
	IT_Databus_c: REAL;
	IT_Databus_o3: REAL;
	IT_Databus_e: REAL;
	IT_Databus_n0: BOOL;
	IT_Databus_ep: BOOL;
	IT_Databus_l: BOOL;
	IT_Databus_f: BOOL;
	IT_Databus_k: BOOL;
	IT_Databus_g: BOOL;
	IT_Databus_b: BOOL;
	IT_Databus_d: BOOL;
	IT_Databus_h: BOOL;
	IT_Databus_j: BOOL;
	IT_Databus_ja: BOOL;
	IT_Databus_if: BOOL;
	FL_BDUControl_Databus: LREAL;
	FL_BDUControl_Databus_o: LREAL;
	FL_BDUControl_Databus_n: LREAL;
	FL_BatteryBox_HVControl_Databus: LREAL;
	FL_BatteryBox_HVControl_Databus_b: LREAL;
	FL_BatteryBox_HVControl_Databus_a: LREAL;
	FL_u8SS_EmergencySD: BOOL;
END_VAR
VAR_OUTPUT
	FL_boSS_System_SD: BOOL;
	FL_u8SS_System_SD_ErrorCode: USINT;
END_VAR
VAR
	is_active_c39_ChiefMaster: USINT;
	is_c39_ChiefMaster: USINT;
	DelayInput1_DSTATE: LREAL;
	DelayInput1_DSTATE_a: LREAL;
	DelayInput1_DSTATE_j: LREAL;
	i0_BDU_Error: BDU_Error;
	i0_Chart_ek: Chart_ek;
	i1_Chart_ek: Chart_ek;
	i2_Chart_ek: Chart_ek;
	i0_IMD_SD: IMD_SD;
	rtb_OR1_c: BOOL;
	rtb_Switch_k: BOOL;
	rtb_FixPtRelationalOperator_h5: BOOL;
	rtb_Out_nh: BOOL;
	rtb_FixPtRelationalOperator_m: BOOL;
	rtb_Out_lz: BOOL;
	rtb_Switch1_j1g: BOOL;
	rtb_Compare_jn: BOOL;
	temp1: DINT;
END_VAR



CASE ssMethodType OF
    SS_INITIALIZE: 
        (* InitializeConditions for UnitDelay: '<S181>/Delay Input1'
         *
         * Block description for '<S181>/Delay Input1':
         *  
         *  Store in Global RAM *)
        DelayInput1_DSTATE := 0.0;
        (* InitializeConditions for UnitDelay: '<S182>/Delay Input1'
         *
         * Block description for '<S182>/Delay Input1':
         *  
         *  Store in Global RAM *)
        DelayInput1_DSTATE_a := 0.0;
        (* InitializeConditions for UnitDelay: '<S183>/Delay Input1'
         *
         * Block description for '<S183>/Delay Input1':
         *  
         *  Store in Global RAM *)
        DelayInput1_DSTATE_j := 0.0;
        i0_BDU_Error(ssMethodType := SS_INITIALIZE, Main_REL_Databus := FL_BDUControl_Databus, Main_REL_Databus_c := FL_BDUControl_Databus_o, Main_REL_Databus_p := FL_BDUControl_Databus_n);
        i0_Chart_ek(ssMethodType := SS_INITIALIZE, In := rtb_FixPtRelationalOperator_h5, REQ_HV_ON_BB := rtb_FixPtRelationalOperator_h5, KL15_CM_Reset := FL_boKL15_Reset);
        rtb_Out_nh := i0_Chart_ek.Out;
        i1_Chart_ek(ssMethodType := SS_INITIALIZE, In := rtb_FixPtRelationalOperator_m, REQ_HV_ON_BB := rtb_FixPtRelationalOperator_m, KL15_CM_Reset := FL_boKL15_Reset);
        rtb_FixPtRelationalOperator_h5 := i1_Chart_ek.Out;
        i2_Chart_ek(ssMethodType := SS_INITIALIZE, In := rtb_FixPtRelationalOperator_m, REQ_HV_ON_BB := rtb_FixPtRelationalOperator_m, KL15_CM_Reset := FL_boKL15_Reset);
        rtb_Out_lz := i2_Chart_ek.Out;
        i0_IMD_SD(ssMethodType := SS_INITIALIZE, BatteryPackSignals := IT_Databus_f, BatteryPackSignals_g := IT_Databus_m, BatteryPackSignals_f := IT_Databus_k, BatteryPackSignals_d := IT_Databus_a, BatteryPackSignals_c := IT_Databus_g, BatteryPackSignals_c4 := IT_Databus_or, BatteryPackSignals_dh := IT_Databus_b, BatteryPackSignals_k := IT_Databus_d, BatteryPackSignals_g5 := IT_Databus_h, BatteryPackSignals_b := IT_Databus_j, BatteryPackSignals_di := IT_Databus_ja, BatteryPackSignals_n := IT_Databus_if);
        (* SystemInitialize for Chart: '<S115>/Chart' *)
        is_active_c39_ChiefMaster := 0;
        is_c39_ChiefMaster := ChiefMaster_IN_NO_ACTIVE_CHILD_cs;
        FL_boSS_System_SD := FALSE;
    SS_OUTPUT: 
        (* RelationalOperator: '<S158>/Compare' incorporates:
         *  Constant: '<S158>/Constant' *)
        rtb_FixPtRelationalOperator_m := IT_Databus = 0;
        (* Switch: '<S164>/Switch' incorporates:
         *  Constant: '<S164>/Constant'
         *  Logic: '<S164>/AND' *)

        IF IT_Databus_m AND rtb_FixPtRelationalOperator_m THEN 
            rtb_Switch_k := IT_Databus_n;
        ELSE 
            rtb_Switch_k := FALSE;
        END_IF;

        (* End of Switch: '<S164>/Switch' *)
        

        (* Switch: '<S163>/Switch1' incorporates:
         *  Constant: '<S163>/Constant'
         *  Logic: '<S163>/AND1' *)

        IF IT_Databus_a AND rtb_FixPtRelationalOperator_m THEN 
            rtb_Switch1_j1g := IT_Databus_o;
        ELSE 
            rtb_Switch1_j1g := FALSE;
        END_IF;

        (* End of Switch: '<S163>/Switch1' *)
        

        (* Switch: '<S162>/Switch2' incorporates:
         *  Constant: '<S162>/Constant'
         *  Logic: '<S162>/AND2' *)

        IF IT_Databus_or AND rtb_FixPtRelationalOperator_m THEN 
            rtb_FixPtRelationalOperator_m := IT_Databus_i;
        ELSE 
            rtb_FixPtRelationalOperator_m := FALSE;
        END_IF;

        (* End of Switch: '<S162>/Switch2' *)
        i0_BDU_Error(ssMethodType := SS_OUTPUT, Main_REL_Databus := FL_BDUControl_Databus, Main_REL_Databus_c := FL_BDUControl_Databus_o, Main_REL_Databus_p := FL_BDUControl_Databus_n);
        rtb_OR1_c := i0_BDU_Error.BDU_Error_lg;
        (* RelationalOperator: '<S181>/FixPt Relational Operator' incorporates:
         *  Constant: '<S176>/Constant'
         *  RelationalOperator: '<S176>/Compare'
         *  UnitDelay: '<S181>/Delay Input1'
         *
         * Block description for '<S181>/Delay Input1':
         *  
         *  Store in Global RAM *)
        i0_Chart_ek(ssMethodType := SS_OUTPUT, In := FL_BatteryBox_HVControl_Databus < DelayInput1_DSTATE, REQ_HV_ON_BB := FL_BatteryBox_HVControl_Databus = 0.0, KL15_CM_Reset := FL_boKL15_Reset);
        rtb_Out_nh := i0_Chart_ek.Out;
        (* RelationalOperator: '<S182>/FixPt Relational Operator' incorporates:
         *  Constant: '<S178>/Constant'
         *  RelationalOperator: '<S178>/Compare'
         *  UnitDelay: '<S182>/Delay Input1'
         *
         * Block description for '<S182>/Delay Input1':
         *  
         *  Store in Global RAM *)
        i1_Chart_ek(ssMethodType := SS_OUTPUT, In := FL_BatteryBox_HVControl_Databus_b < DelayInput1_DSTATE_a, REQ_HV_ON_BB := FL_BatteryBox_HVControl_Databus_b = 0.0, KL15_CM_Reset := FL_boKL15_Reset);
        rtb_FixPtRelationalOperator_h5 := i1_Chart_ek.Out;
        (* RelationalOperator: '<S183>/FixPt Relational Operator' incorporates:
         *  Constant: '<S180>/Constant'
         *  RelationalOperator: '<S180>/Compare'
         *  UnitDelay: '<S183>/Delay Input1'
         *
         * Block description for '<S183>/Delay Input1':
         *  
         *  Store in Global RAM *)
        i2_Chart_ek(ssMethodType := SS_OUTPUT, In := FL_BatteryBox_HVControl_Databus_a < DelayInput1_DSTATE_j, REQ_HV_ON_BB := FL_BatteryBox_HVControl_Databus_a = 0.0, KL15_CM_Reset := FL_boKL15_Reset);
        rtb_Out_lz := i2_Chart_ek.Out;
        (* Logic: '<S161>/OR' incorporates:
         *  Constant: '<S175>/Constant'
         *  Constant: '<S177>/Constant'
         *  Constant: '<S179>/Constant'
         *  Logic: '<S161>/AND'
         *  Logic: '<S161>/AND1'
         *  Logic: '<S161>/AND2'
         *  RelationalOperator: '<S175>/Compare'
         *  RelationalOperator: '<S177>/Compare'
         *  RelationalOperator: '<S179>/Compare' *)
        rtb_FixPtRelationalOperator_h5 := ((((IT_Databus_c > 1.0) AND IT_Databus_n) AND rtb_Out_nh) OR (((IT_Databus_o3 > 1.0) AND IT_Databus_o) AND rtb_FixPtRelationalOperator_h5)) OR (((IT_Databus_e > 1.0) AND IT_Databus_i) AND rtb_Out_lz);
        rtb_Out_lz := IMD_Error(BatteryPackSignals := IT_Databus_f, BatteryPackSignals_l := IT_Databus_m, BatteryPackSignals_d := IT_Databus_k, BatteryPackSignals_n := IT_Databus_a, BatteryPackSignals_f := IT_Databus_g, BatteryPackSignals_dk := IT_Databus_or);
        i0_IMD_SD(ssMethodType := SS_OUTPUT, BatteryPackSignals := IT_Databus_f, BatteryPackSignals_g := IT_Databus_m, BatteryPackSignals_f := IT_Databus_k, BatteryPackSignals_d := IT_Databus_a, BatteryPackSignals_c := IT_Databus_g, BatteryPackSignals_c4 := IT_Databus_or, BatteryPackSignals_dh := IT_Databus_b, BatteryPackSignals_k := IT_Databus_d, BatteryPackSignals_g5 := IT_Databus_h, BatteryPackSignals_b := IT_Databus_j, BatteryPackSignals_di := IT_Databus_ja, BatteryPackSignals_n := IT_Databus_if);
        rtb_Out_nh := i0_IMD_SD.IMD_SDError;
        (* Logic: '<S165>/AND3' incorporates:
         *  RelationalOperator: '<S184>/Compare'
         *  RelationalOperator: '<S185>/Compare'
         *  RelationalOperator: '<S186>/Compare' *)
        rtb_Compare_jn := (( NOT IT_Databus_n0) OR ( NOT IT_Databus_ep)) OR ( NOT IT_Databus_l);
        (* Sum: '<S115>/Add' incorporates:
         *  Gain: '<S115>/Gain'
         *  Gain: '<S115>/Gain1'
         *  Gain: '<S115>/Gain2'
         *  Gain: '<S115>/Gain3'
         *  Gain: '<S115>/Gain4'
         *  Gain: '<S115>/Gain5'
         *  Gain: '<S115>/Gain6'
         *  Gain: '<S115>/Gain7'
         *  Gain: '<S115>/Gain8' *)

        IF FL_u8SS_EmergencySD THEN 
            temp1 := 255;
        ELSE 
            temp1 := 0;
        END_IF;

        FL_u8SS_System_SD_ErrorCode := UDINT_TO_USINT(DWORD_TO_UDINT(SHR(UDINT_TO_DWORD((((((((DWORD_TO_UDINT(SHL(UDINT_TO_DWORD(USINT_TO_UDINT(DINT_TO_USINT(DWORD_TO_DINT(SHL(DINT_TO_DWORD(BOOL_TO_DINT(rtb_Switch1_j1g)), 7))))), 1)) + USINT_TO_UDINT(DINT_TO_USINT(DWORD_TO_DINT(SHL(DINT_TO_DWORD(BOOL_TO_DINT(rtb_Switch_k)), 7))))) + DWORD_TO_UDINT(SHL(UDINT_TO_DWORD(USINT_TO_UDINT(DINT_TO_USINT(DWORD_TO_DINT(SHL(DINT_TO_DWORD(BOOL_TO_DINT(rtb_FixPtRelationalOperator_m)), 7))))), 2))) + DWORD_TO_UDINT(SHL(UDINT_TO_DWORD(USINT_TO_UDINT(DINT_TO_USINT(DWORD_TO_DINT(SHL(DINT_TO_DWORD(BOOL_TO_DINT(rtb_OR1_c)), 7))))), 3))) + DWORD_TO_UDINT(SHL(UDINT_TO_DWORD(DINT_TO_UDINT(DWORD_TO_DINT(SHL(DINT_TO_DWORD(BOOL_TO_DINT(rtb_FixPtRelationalOperator_h5)), 7)))), 4))) + DWORD_TO_UDINT(SHL(UDINT_TO_DWORD(DINT_TO_UDINT(DWORD_TO_DINT(SHL(DINT_TO_DWORD(BOOL_TO_DINT(rtb_Out_lz)), 7)))), 5))) + DWORD_TO_UDINT(SHL(UDINT_TO_DWORD(DINT_TO_UDINT(DWORD_TO_DINT(SHL(DINT_TO_DWORD(BOOL_TO_DINT(rtb_Out_nh)), 7)))), 6))) + DWORD_TO_UDINT(SHL(UDINT_TO_DWORD(DINT_TO_UDINT(DWORD_TO_DINT(SHL(DINT_TO_DWORD(BOOL_TO_DINT(rtb_Compare_jn)), 7)))), 7))) + DWORD_TO_UDINT(SHL(UDINT_TO_DWORD(DINT_TO_UDINT(temp1)), 7))), 7)));
        (* Chart: '<S115>/Chart' incorporates:
         *  Logic: '<S115>/OR' *)
        (* Gateway: ChiefMaster/Flow Logic/System Status/SDError/Chart *)
        (* During: ChiefMaster/Flow Logic/System Status/SDError/Chart *)

        IF is_active_c39_ChiefMaster = 0 THEN 
            (* Entry: ChiefMaster/Flow Logic/System Status/SDError/Chart *)
            is_active_c39_ChiefMaster := 1;
            (* Entry Internal: ChiefMaster/Flow Logic/System Status/SDError/Chart *)
            (* Transition: '<S157>:4' *)
            is_c39_ChiefMaster := ChiefMaster_IN_Default_fd;
            (* Entry 'Default': '<S157>:3' *)
            (* '<S157>:3:2' System_Error = false; *)
            FL_boSS_System_SD := FALSE;
        ELSE 

            CASE is_c39_ChiefMaster OF
                ChiefMaster_IN_Default_fd: 
                    (* During 'Default': '<S157>:3' *)
                    (* '<S157>:7:1' sf_internal_predicateOutput = In == true; *)

                    IF ((((((rtb_Switch_k OR rtb_Switch1_j1g) OR rtb_FixPtRelationalOperator_m) OR rtb_OR1_c) OR rtb_FixPtRelationalOperator_h5) OR rtb_Out_lz) OR rtb_Compare_jn) OR FL_u8SS_EmergencySD THEN 
                        (* Transition: '<S157>:7' *)
                        is_c39_ChiefMaster := ChiefMaster_IN_Error_ex;
                        (* Entry 'Error': '<S157>:6' *)
                        (* '<S157>:6:2' System_Error = true; *)
                        FL_boSS_System_SD := TRUE;
                    ELSE 
                        (* '<S157>:3:2' System_Error = false; *)
                        FL_boSS_System_SD := FALSE;
                    END_IF;

                ELSE
                    (* During 'Error': '<S157>:6' *)
                    (* '<S157>:9:1' sf_internal_predicateOutput = KL15_CM_reset == true; *)

                    IF FL_boKL15_Reset THEN 
                        (* Transition: '<S157>:9' *)
                        is_c39_ChiefMaster := ChiefMaster_IN_Default_fd;
                        (* Entry 'Default': '<S157>:3' *)
                        (* '<S157>:3:2' System_Error = false; *)
                        FL_boSS_System_SD := FALSE;
                    ELSE 
                        (* '<S157>:6:2' System_Error = true; *)
                        FL_boSS_System_SD := TRUE;
                    END_IF;

            END_CASE;

        END_IF;

        (* End of Chart: '<S115>/Chart' *)
    SS_UPDATE: 
        i0_BDU_Error(ssMethodType := SS_UPDATE, Main_REL_Databus := FL_BDUControl_Databus, Main_REL_Databus_c := FL_BDUControl_Databus_o, Main_REL_Databus_p := FL_BDUControl_Databus_n);
        rtb_OR1_c := i0_BDU_Error.BDU_Error_lg;
        (* Update for UnitDelay: '<S181>/Delay Input1'
         *
         * Block description for '<S181>/Delay Input1':
         *  
         *  Store in Global RAM *)
        DelayInput1_DSTATE := FL_BatteryBox_HVControl_Databus;
        (* Update for UnitDelay: '<S182>/Delay Input1'
         *
         * Block description for '<S182>/Delay Input1':
         *  
         *  Store in Global RAM *)
        DelayInput1_DSTATE_a := FL_BatteryBox_HVControl_Databus_b;
        (* Update for UnitDelay: '<S183>/Delay Input1'
         *
         * Block description for '<S183>/Delay Input1':
         *  
         *  Store in Global RAM *)
        DelayInput1_DSTATE_j := FL_BatteryBox_HVControl_Databus_a;
END_CASE;

END_FUNCTION_BLOCK

// Device/Application/IMD_Error
FUNCTION IMD_Error : BOOL
VAR_INPUT
	BatteryPackSignals: BOOL;
	BatteryPackSignals_l: BOOL;
	BatteryPackSignals_d: BOOL;
	BatteryPackSignals_n: BOOL;
	BatteryPackSignals_f: BOOL;
	BatteryPackSignals_dk: BOOL;
END_VAR
VAR
END_VAR


(* RelationalOperator: '<S159>/GreaterThan' incorporates:
 *  Constant: '<S159>/Constant'
 *  Logic: '<S159>/AND1'
 *  Logic: '<S159>/AND2'
 *  Logic: '<S159>/AND3'
 *  Sum: '<S159>/Sum' *)
IMD_Error := ((BOOL_TO_UDINT(BatteryPackSignals AND BatteryPackSignals_l) + BOOL_TO_UDINT(BatteryPackSignals_d AND BatteryPackSignals_n)) + BOOL_TO_UDINT(BatteryPackSignals_f AND BatteryPackSignals_dk)) > 1;

END_FUNCTION

// Device/Application/BDU_Error
FUNCTION_BLOCK BDU_Error
VAR_INPUT
	ssMethodType: SINT;
	Main_REL_Databus: LREAL;
	Main_REL_Databus_c: LREAL;
	Main_REL_Databus_p: LREAL;
END_VAR
VAR_OUTPUT
	BDU_Error_lg: BOOL;
END_VAR
VAR
	UnitDelay_DSTATE: LREAL;
	UnitDelay1_DSTATE: LREAL;
	UnitDelay2_DSTATE: LREAL;
END_VAR



CASE ssMethodType OF
    SS_INITIALIZE: 
        (* InitializeConditions for UnitDelay: '<S156>/Unit Delay' *)
        UnitDelay_DSTATE := 0.0;
        (* InitializeConditions for UnitDelay: '<S156>/Unit Delay1' *)
        UnitDelay1_DSTATE := 0.0;
        (* InitializeConditions for UnitDelay: '<S156>/Unit Delay2' *)
        UnitDelay2_DSTATE := 0.0;
    SS_OUTPUT: 
        (* Logic: '<S156>/OR1' incorporates:
         *  Constant: '<S166>/Constant'
         *  Constant: '<S167>/Constant'
         *  Constant: '<S168>/Constant'
         *  RelationalOperator: '<S166>/Compare'
         *  RelationalOperator: '<S167>/Compare'
         *  RelationalOperator: '<S168>/Compare'
         *  UnitDelay: '<S156>/Unit Delay'
         *  UnitDelay: '<S156>/Unit Delay1'
         *  UnitDelay: '<S156>/Unit Delay2' *)
        BDU_Error_lg := ((UnitDelay_DSTATE = 3.0) OR (UnitDelay1_DSTATE = 3.0)) OR (UnitDelay2_DSTATE = 2.0);
    SS_UPDATE: 
        (* Update for UnitDelay: '<S156>/Unit Delay' *)
        UnitDelay_DSTATE := Main_REL_Databus;
        (* Update for UnitDelay: '<S156>/Unit Delay1' *)
        UnitDelay1_DSTATE := Main_REL_Databus_c;
        (* Update for UnitDelay: '<S156>/Unit Delay2' *)
        UnitDelay2_DSTATE := Main_REL_Databus_p;
END_CASE;

END_FUNCTION_BLOCK

// Device/Application/Chart_ek
FUNCTION_BLOCK Chart_ek
VAR_INPUT
	ssMethodType: SINT;
	In: BOOL;
	REQ_HV_ON_BB: BOOL;
	KL15_CM_Reset: BOOL;
END_VAR
VAR_OUTPUT
	Out: BOOL;
END_VAR
VAR
	is_active_c42_ChiefMaster: USINT;
	is_c42_ChiefMaster: USINT;
	temporalCounter_i1: PLC_CODER_TIMER;
END_VAR



CASE ssMethodType OF
    SS_INITIALIZE: 
        temporalCounter_i1(timerAction := 1, maxTime := 0);
        is_active_c42_ChiefMaster := 0;
        is_c42_ChiefMaster := ChiefMaster_IN_NO_ACTIVE_CHILD_ir;
        Out := FALSE;
    SS_OUTPUT: 
        (* Chart: '<S161>/Chart' *)
        (* Gateway: ChiefMaster/Flow Logic/System Status/SDError/Subsystem/Chart *)
        (* During: ChiefMaster/Flow Logic/System Status/SDError/Subsystem/Chart *)

        IF is_active_c42_ChiefMaster = 0 THEN 
            (* Entry: ChiefMaster/Flow Logic/System Status/SDError/Subsystem/Chart *)
            is_active_c42_ChiefMaster := 1;
            (* Entry Internal: ChiefMaster/Flow Logic/System Status/SDError/Subsystem/Chart *)
            (* Transition: '<S172>:2' *)
            is_c42_ChiefMaster := ChiefMaster_IN_Default_h3;
            (* Entry 'Default': '<S172>:1' *)
            (* '<S172>:1:2' Out = false *)
            Out := FALSE;
        ELSE 

            CASE is_c42_ChiefMaster OF
                ChiefMaster_IN_Actual_e: 
                    (* During 'Actual': '<S172>:3' *)
                    (* '<S172>:15:1' sf_internal_predicateOutput = KL15_CM_Reset == true; *)

                    IF KL15_CM_Reset THEN 
                        (* Transition: '<S172>:15' *)
                        is_c42_ChiefMaster := ChiefMaster_IN_Default_h3;
                        (* Entry 'Default': '<S172>:1' *)
                        (* '<S172>:1:2' Out = false *)
                        Out := FALSE;
                    ELSE 
                        (* '<S172>:3:2' Out = REQ_HV_ON_BB *)
                        Out := REQ_HV_ON_BB;
                    END_IF;

                ChiefMaster_IN_Default_h3: 
                    (* During 'Default': '<S172>:1' *)
                    (* '<S172>:4:1' sf_internal_predicateOutput = In == true; *)

                    IF In THEN 
                        (* Transition: '<S172>:4' *)
                        is_c42_ChiefMaster := ChiefMaster_IN_hold_n;
                        temporalCounter_i1(timerAction := 1, maxTime := 0);
                        (* Entry 'hold': '<S172>:7' *)
                        (* '<S172>:7:2' Out = false *)
                        Out := FALSE;
                    ELSE 
                        (* '<S172>:1:2' Out = false *)
                        Out := FALSE;
                    END_IF;

                ELSE
                    (* During 'hold': '<S172>:7' *)
                    (* '<S172>:8:1' sf_internal_predicateOutput = after(5,sec); *)
                    temporalCounter_i1(timerAction := 2, maxTime := 5000);

                    IF temporalCounter_i1.done THEN 
                        (* Transition: '<S172>:8' *)
                        is_c42_ChiefMaster := ChiefMaster_IN_Actual_e;
                        (* Entry 'Actual': '<S172>:3' *)
                        (* '<S172>:3:2' Out = REQ_HV_ON_BB *)
                        Out := REQ_HV_ON_BB;
                    ELSE 
                        (* '<S172>:7:2' Out = false *)
                        Out := FALSE;
                    END_IF;

            END_CASE;

        END_IF;

        (* End of Chart: '<S161>/Chart' *)
END_CASE;

END_FUNCTION_BLOCK

// Device/Application/IMD_SD
FUNCTION_BLOCK IMD_SD
VAR_INPUT
	ssMethodType: SINT;
	BatteryPackSignals: BOOL;
	BatteryPackSignals_g: BOOL;
	BatteryPackSignals_f: BOOL;
	BatteryPackSignals_d: BOOL;
	BatteryPackSignals_c: BOOL;
	BatteryPackSignals_c4: BOOL;
	BatteryPackSignals_dh: BOOL;
	BatteryPackSignals_k: BOOL;
	BatteryPackSignals_g5: BOOL;
	BatteryPackSignals_b: BOOL;
	BatteryPackSignals_di: BOOL;
	BatteryPackSignals_n: BOOL;
END_VAR
VAR_OUTPUT
	IMD_SDError: BOOL;
END_VAR
VAR
	i0_Chart_ls: Chart_ls;
	i1_Chart_ls: Chart_ls;
	i2_Chart_ls: Chart_ls;
	rtb_IMD_Error_k: BOOL;
	rtb_IMD_Error_i: BOOL;
	rtb_IMD_Error: BOOL;
END_VAR



CASE ssMethodType OF
    SS_INITIALIZE: 
        i0_Chart_ls(ssMethodType := SS_INITIALIZE, IP_boBMS_InsulationReadyOK := BatteryPackSignals_dh, IP_boBMS_InsulationSDError := BatteryPackSignals_k);
        rtb_IMD_Error_k := i0_Chart_ls.IMD_Error_l;
        i1_Chart_ls(ssMethodType := SS_INITIALIZE, IP_boBMS_InsulationReadyOK := BatteryPackSignals_g5, IP_boBMS_InsulationSDError := BatteryPackSignals_b);
        rtb_IMD_Error_i := i1_Chart_ls.IMD_Error_l;
        i2_Chart_ls(ssMethodType := SS_INITIALIZE, IP_boBMS_InsulationReadyOK := BatteryPackSignals_di, IP_boBMS_InsulationSDError := BatteryPackSignals_n);
        rtb_IMD_Error := i2_Chart_ls.IMD_Error_l;
    SS_OUTPUT: 
        i0_Chart_ls(ssMethodType := SS_OUTPUT, IP_boBMS_InsulationReadyOK := BatteryPackSignals_dh, IP_boBMS_InsulationSDError := BatteryPackSignals_k);
        rtb_IMD_Error_k := i0_Chart_ls.IMD_Error_l;
        i1_Chart_ls(ssMethodType := SS_OUTPUT, IP_boBMS_InsulationReadyOK := BatteryPackSignals_g5, IP_boBMS_InsulationSDError := BatteryPackSignals_b);
        rtb_IMD_Error_i := i1_Chart_ls.IMD_Error_l;
        i2_Chart_ls(ssMethodType := SS_OUTPUT, IP_boBMS_InsulationReadyOK := BatteryPackSignals_di, IP_boBMS_InsulationSDError := BatteryPackSignals_n);
        rtb_IMD_Error := i2_Chart_ls.IMD_Error_l;
        (* Logic: '<S160>/OR' incorporates:
         *  Logic: '<S160>/AND'
         *  Logic: '<S160>/AND1'
         *  Logic: '<S160>/AND2' *)
        IMD_SDError := (((rtb_IMD_Error_k AND BatteryPackSignals) AND BatteryPackSignals_g) OR ((rtb_IMD_Error_i AND BatteryPackSignals_f) AND BatteryPackSignals_d)) OR ((rtb_IMD_Error AND BatteryPackSignals_c) AND BatteryPackSignals_c4);
END_CASE;

END_FUNCTION_BLOCK

// Device/Application/Chart_ls
FUNCTION_BLOCK Chart_ls
VAR_INPUT
	ssMethodType: SINT;
	IP_boBMS_InsulationReadyOK: BOOL;
	IP_boBMS_InsulationSDError: BOOL;
END_VAR
VAR_OUTPUT
	IMD_Error_l: BOOL;
END_VAR
VAR
	is_active_c24_ChiefMaster: USINT;
	is_c24_ChiefMaster: USINT;
END_VAR



CASE ssMethodType OF
    SS_INITIALIZE: 
        is_active_c24_ChiefMaster := 0;
        is_c24_ChiefMaster := ChiefMaster_IN_NO_ACTIVE_CHILD_eq;
        IMD_Error_l := FALSE;
    SS_OUTPUT: 
        (* Chart: '<S160>/Chart' *)
        (* Gateway: ChiefMaster/Flow Logic/System Status/SDError/IMD_SD/Chart *)
        (* During: ChiefMaster/Flow Logic/System Status/SDError/IMD_SD/Chart *)

        IF is_active_c24_ChiefMaster = 0 THEN 
            (* Entry: ChiefMaster/Flow Logic/System Status/SDError/IMD_SD/Chart *)
            is_active_c24_ChiefMaster := 1;
            (* Entry Internal: ChiefMaster/Flow Logic/System Status/SDError/IMD_SD/Chart *)
            (* Transition: '<S169>:3' *)
            is_c24_ChiefMaster := ChiefMaster_IN_Default_jp;
            (* Entry 'Default': '<S169>:2' *)
            (* '<S169>:2:2' IMD_Error=false; *)
            IMD_Error_l := FALSE;
        ELSE 

            CASE is_c24_ChiefMaster OF
                ChiefMaster_IN_Default_jp: 
                    (* During 'Default': '<S169>:2' *)
                    (* '<S169>:5:1' sf_internal_predicateOutput = IP_boBMS_InsulationReadyOK == true; *)

                    IF IP_boBMS_InsulationReadyOK THEN 
                        (* Transition: '<S169>:5' *)
                        is_c24_ChiefMaster := ChiefMaster_IN_IsoMonitorCheck;
                        (* Entry 'IsoMonitorCheck': '<S169>:4' *)
                        (* '<S169>:4:2' IMD_Error=false; *)
                        IMD_Error_l := FALSE;
                    ELSE 
                        (* '<S169>:2:2' IMD_Error=false; *)
                        IMD_Error_l := FALSE;
                    END_IF;

                ChiefMaster_IN_IsoMonitorCheck: 
                    (* During 'IsoMonitorCheck': '<S169>:4' *)
                    (* '<S169>:8:1' sf_internal_predicateOutput = IP_boBMS_InsulationSDError == true; *)

                    IF IP_boBMS_InsulationSDError THEN 
                        (* Transition: '<S169>:8' *)
                        is_c24_ChiefMaster := ChiefMaster_IN_IsoMonitorError;
                        (* Entry 'IsoMonitorError': '<S169>:7' *)
                        (* '<S169>:7:2' IMD_Error=true; *)
                        IMD_Error_l := TRUE;
                    ELSE 
                        (* '<S169>:4:2' IMD_Error=false; *)
                        IMD_Error_l := FALSE;
                    END_IF;

                ELSE
                    (* During 'IsoMonitorError': '<S169>:7' *)
                    (* '<S169>:7:2' IMD_Error=true; *)
                    IMD_Error_l := TRUE;
            END_CASE;

        END_IF;

        (* End of Chart: '<S160>/Chart' *)
END_CASE;

END_FUNCTION_BLOCK

// Device/Application/BattChargeFcn
FUNCTION_BLOCK BattChargeFcn
VAR_INPUT
	ssMethodType: SINT;
	MaxChargeCurr_fb: REAL;
	MaxChargeCurrentBatt: REAL;
	ChargeStopPressed: BOOL;
	HV_ON_Batt1: BOOL;
	HV_ON_Batt2: BOOL;
	HV_ON_Batt3: BOOL;
	Ibatt1: REAL;
	Ibatt2: REAL;
	Ibatt3: REAL;
	Fcn_available: BOOL;
	CurrentReductionConstant: REAL;
	CurrentLB_f: REAL;
	CurrentUB_c: REAL;
END_VAR
VAR_OUTPUT
	FL_sST_MaxChargeCurrent: REAL;
	REQ_HV_Open_Batt2: BOOL;
	REQ_HV_Open_Batt3: BOOL;
	REQ_HV_Open_Batt1: BOOL;
	BatteryReadyToShutDown: BOOL;
END_VAR
VAR
	temporalCounter_i1: PLC_CODER_TIMER;
	is_c52_ChiefMaster: USINT;
	is_active_c52_ChiefMaster: USINT;
	temp1: BOOL;
END_VAR



CASE ssMethodType OF
    SS_INITIALIZE: 
        temporalCounter_i1(timerAction := 1, maxTime := 0);
        is_active_c52_ChiefMaster := 0;
        is_c52_ChiefMaster := ChiefMaster_IN_NO_ACTIVE_CHILD_c;
        FL_sST_MaxChargeCurrent := 0.0;
        REQ_HV_Open_Batt2 := FALSE;
        REQ_HV_Open_Batt3 := FALSE;
        REQ_HV_Open_Batt1 := FALSE;
        BatteryReadyToShutDown := FALSE;
    SS_OUTPUT: 
        (* Chart: '<S110>/BattChargeFcn' *)
        (* Gateway: ChiefMaster/Flow Logic/System Status/CurrentPrognosis/BattChargeFcn *)
        (* During: ChiefMaster/Flow Logic/System Status/CurrentPrognosis/BattChargeFcn *)

        IF is_active_c52_ChiefMaster = 0 THEN 
            (* Entry: ChiefMaster/Flow Logic/System Status/CurrentPrognosis/BattChargeFcn *)
            is_active_c52_ChiefMaster := 1;
            (* Entry Internal: ChiefMaster/Flow Logic/System Status/CurrentPrognosis/BattChargeFcn *)
            (* Transition: '<S125>:5' *)
            is_c52_ChiefMaster := ChiefMaster_IN_Default_b0;
            (* Entry 'Default': '<S125>:4' *)
            (* '<S125>:4:2' FL_sST_MaxChargeCurrent = MaxChargeCurrentBatt *)
            FL_sST_MaxChargeCurrent := MaxChargeCurrentBatt;
            (* '<S125>:4:3' REQ_HV_Open_Batt1 = false *)
            REQ_HV_Open_Batt1 := FALSE;
            (* '<S125>:4:4' REQ_HV_Open_Batt2 = false *)
            REQ_HV_Open_Batt2 := FALSE;
            (* '<S125>:4:5' REQ_HV_Open_Batt3 = false *)
            REQ_HV_Open_Batt3 := FALSE;
            (* '<S125>:4:6' BatteryReadyToShutDown = true *)
            BatteryReadyToShutDown := TRUE;
        ELSE 

            CASE is_c52_ChiefMaster OF
                ChiefMaster_IN_Batt1: 
                    (* During 'Batt1': '<S125>:11' *)
                    (* '<S125>:14:1' sf_internal_predicateOutput = HV_ON_Batt1 == 0 ||... *)
                    (* '<S125>:14:2' after(20,sec); *)
                    temp1 := FALSE;

                    IF  NOT HV_ON_Batt1 THEN 
                        temp1 := TRUE;
                    ELSE 
                        temporalCounter_i1(timerAction := 2, maxTime := 20000);

                        IF temporalCounter_i1.done THEN 
                            temp1 := TRUE;
                        ELSE 
                            (* '<S125>:11:2' REQ_HV_Open_Batt1 = true *)
                            REQ_HV_Open_Batt1 := TRUE;
                        END_IF;

                    END_IF;


                    IF temp1 THEN 
                        (* Transition: '<S125>:14' *)
                        is_c52_ChiefMaster := ChiefMaster_IN_RampDown;
                        (* Entry 'RampDown': '<S125>:6' *)
                        (* '<S125>:6:2' FL_sST_MaxChargeCurrent = (FL_sST_MaxChargeCurrent - CurrentReductionConstant) *)
                        FL_sST_MaxChargeCurrent := FL_sST_MaxChargeCurrent - CurrentReductionConstant;
                        (* '<S125>:6:3' REQ_HV_Open_Batt1 = false *)
                        REQ_HV_Open_Batt1 := FALSE;
                        (* '<S125>:6:4' REQ_HV_Open_Batt2 = false *)
                        REQ_HV_Open_Batt2 := FALSE;
                        (* '<S125>:6:5' REQ_HV_Open_Batt3 = false *)
                        REQ_HV_Open_Batt3 := FALSE;
                        (* '<S125>:6:6' BatteryReadyToShutDown = false *)
                        BatteryReadyToShutDown := FALSE;
                    END_IF;

                ChiefMaster_IN_Batt2: 
                    (* During 'Batt2': '<S125>:18' *)
                    (* '<S125>:17:1' sf_internal_predicateOutput = HV_ON_Batt2 == 0 ||... *)
                    (* '<S125>:17:2' after(20,sec); *)
                    temp1 := FALSE;

                    IF  NOT HV_ON_Batt2 THEN 
                        temp1 := TRUE;
                    ELSE 
                        temporalCounter_i1(timerAction := 2, maxTime := 20000);

                        IF temporalCounter_i1.done THEN 
                            temp1 := TRUE;
                        ELSE 
                            (* '<S125>:18:2' REQ_HV_Open_Batt2 = true *)
                            REQ_HV_Open_Batt2 := TRUE;
                        END_IF;

                    END_IF;


                    IF temp1 THEN 
                        (* Transition: '<S125>:17' *)
                        is_c52_ChiefMaster := ChiefMaster_IN_RampDown;
                        (* Entry 'RampDown': '<S125>:6' *)
                        (* '<S125>:6:2' FL_sST_MaxChargeCurrent = (FL_sST_MaxChargeCurrent - CurrentReductionConstant) *)
                        FL_sST_MaxChargeCurrent := FL_sST_MaxChargeCurrent - CurrentReductionConstant;
                        (* '<S125>:6:3' REQ_HV_Open_Batt1 = false *)
                        REQ_HV_Open_Batt1 := FALSE;
                        (* '<S125>:6:4' REQ_HV_Open_Batt2 = false *)
                        REQ_HV_Open_Batt2 := FALSE;
                        (* '<S125>:6:5' REQ_HV_Open_Batt3 = false *)
                        REQ_HV_Open_Batt3 := FALSE;
                        (* '<S125>:6:6' BatteryReadyToShutDown = false *)
                        BatteryReadyToShutDown := FALSE;
                    END_IF;

                ChiefMaster_IN_Batt3: 
                    (* During 'Batt3': '<S125>:20' *)
                    (* '<S125>:21:1' sf_internal_predicateOutput = HV_ON_Batt3 == 0 ||... *)
                    (* '<S125>:21:2' after(20,sec); *)
                    temp1 := FALSE;

                    IF  NOT HV_ON_Batt3 THEN 
                        temp1 := TRUE;
                    ELSE 
                        temporalCounter_i1(timerAction := 2, maxTime := 20000);

                        IF temporalCounter_i1.done THEN 
                            temp1 := TRUE;
                        ELSE 
                            (* '<S125>:20:2' REQ_HV_Open_Batt3 = true *)
                            REQ_HV_Open_Batt3 := TRUE;
                        END_IF;

                    END_IF;


                    IF temp1 THEN 
                        (* Transition: '<S125>:21' *)
                        is_c52_ChiefMaster := ChiefMaster_IN_RampDown;
                        (* Entry 'RampDown': '<S125>:6' *)
                        (* '<S125>:6:2' FL_sST_MaxChargeCurrent = (FL_sST_MaxChargeCurrent - CurrentReductionConstant) *)
                        FL_sST_MaxChargeCurrent := FL_sST_MaxChargeCurrent - CurrentReductionConstant;
                        (* '<S125>:6:3' REQ_HV_Open_Batt1 = false *)
                        REQ_HV_Open_Batt1 := FALSE;
                        (* '<S125>:6:4' REQ_HV_Open_Batt2 = false *)
                        REQ_HV_Open_Batt2 := FALSE;
                        (* '<S125>:6:5' REQ_HV_Open_Batt3 = false *)
                        REQ_HV_Open_Batt3 := FALSE;
                        (* '<S125>:6:6' BatteryReadyToShutDown = false *)
                        BatteryReadyToShutDown := FALSE;
                    END_IF;

                ChiefMaster_IN_Default_b0: 
                    (* During 'Default': '<S125>:4' *)
                    (* '<S125>:7:1' sf_internal_predicateOutput = ChargeStopPressed == true &&... *)
                    (* '<S125>:7:2' Fcn_available == true; *)

                    IF ChargeStopPressed AND Fcn_available THEN 
                        (* Transition: '<S125>:7' *)
                        is_c52_ChiefMaster := ChiefMaster_IN_RampDown;
                        (* Entry 'RampDown': '<S125>:6' *)
                        (* '<S125>:6:2' FL_sST_MaxChargeCurrent = (FL_sST_MaxChargeCurrent - CurrentReductionConstant) *)
                        FL_sST_MaxChargeCurrent := FL_sST_MaxChargeCurrent - CurrentReductionConstant;
                        (* '<S125>:6:3' REQ_HV_Open_Batt1 = false *)
                        REQ_HV_Open_Batt1 := FALSE;
                        (* '<S125>:6:4' REQ_HV_Open_Batt2 = false *)
                        REQ_HV_Open_Batt2 := FALSE;
                        (* '<S125>:6:5' REQ_HV_Open_Batt3 = false *)
                        REQ_HV_Open_Batt3 := FALSE;
                        (* '<S125>:6:6' BatteryReadyToShutDown = false *)
                        BatteryReadyToShutDown := FALSE;
                    ELSE 
                        (* '<S125>:4:2' FL_sST_MaxChargeCurrent = MaxChargeCurrentBatt *)
                        FL_sST_MaxChargeCurrent := MaxChargeCurrentBatt;
                        (* '<S125>:4:3' REQ_HV_Open_Batt1 = false *)
                        REQ_HV_Open_Batt1 := FALSE;
                        (* '<S125>:4:4' REQ_HV_Open_Batt2 = false *)
                        REQ_HV_Open_Batt2 := FALSE;
                        (* '<S125>:4:5' REQ_HV_Open_Batt3 = false *)
                        REQ_HV_Open_Batt3 := FALSE;
                        (* '<S125>:4:6' BatteryReadyToShutDown = true *)
                        BatteryReadyToShutDown := TRUE;
                    END_IF;

                ChiefMaster_IN_RampDown: 
                    (* During 'RampDown': '<S125>:6' *)
                    (* '<S125>:12:1' sf_internal_predicateOutput = HV_ON_Batt1 == 1 &&... *)
                    (* '<S125>:12:2' Ibatt1 <= CurrentUB; *)

                    IF HV_ON_Batt1 AND (Ibatt1 <= CurrentUB_c) THEN 
                        (* Transition: '<S125>:12' *)
                        is_c52_ChiefMaster := ChiefMaster_IN_Batt1;
                        temporalCounter_i1(timerAction := 1, maxTime := 0);
                        (* Entry 'Batt1': '<S125>:11' *)
                        (* '<S125>:11:2' REQ_HV_Open_Batt1 = true *)
                        REQ_HV_Open_Batt1 := TRUE;
                    ELSE 
                        (* '<S125>:30:1' sf_internal_predicateOutput = MaxChargeCurr_fb <= 0; *)

                        IF MaxChargeCurr_fb <= 0.0 THEN 
                            (* Transition: '<S125>:30' *)
                            is_c52_ChiefMaster := ChiefMaster_IN_Stop;
                            (* Entry 'Stop': '<S125>:29' *)
                            (* '<S125>:29:2' FL_sST_MaxChargeCurrent = 0; *)
                            FL_sST_MaxChargeCurrent := 0.0;
                            (* '<S125>:29:3' BatteryReadyToShutDown = true *)
                            BatteryReadyToShutDown := TRUE;
                        ELSE 
                            (* '<S125>:19:1' sf_internal_predicateOutput = HV_ON_Batt3 == 1 &&... *)
                            (* '<S125>:19:2' Ibatt3 <= CurrentUB; *)

                            IF HV_ON_Batt3 AND (Ibatt3 <= CurrentUB_c) THEN 
                                (* Transition: '<S125>:19' *)
                                is_c52_ChiefMaster := ChiefMaster_IN_Batt3;
                                temporalCounter_i1(timerAction := 1, maxTime := 0);
                                (* Entry 'Batt3': '<S125>:20' *)
                                (* '<S125>:20:2' REQ_HV_Open_Batt3 = true *)
                                REQ_HV_Open_Batt3 := TRUE;
                            ELSE 
                                (* '<S125>:16:1' sf_internal_predicateOutput = HV_ON_Batt2 == 1 &&... *)
                                (* '<S125>:16:2' Ibatt2 <= CurrentUB; *)

                                IF HV_ON_Batt2 AND (Ibatt2 <= CurrentUB_c) THEN 
                                    (* Transition: '<S125>:16' *)
                                    is_c52_ChiefMaster := ChiefMaster_IN_Batt2;
                                    temporalCounter_i1(timerAction := 1, maxTime := 0);
                                    (* Entry 'Batt2': '<S125>:18' *)
                                    (* '<S125>:18:2' REQ_HV_Open_Batt2 = true *)
                                    REQ_HV_Open_Batt2 := TRUE;
                                ELSE 
                                    (* '<S125>:41:1' sf_internal_predicateOutput = Fcn_available == false; *)

                                    IF  NOT Fcn_available THEN 
                                        (* Transition: '<S125>:41' *)
                                        is_c52_ChiefMaster := ChiefMaster_IN_Default_b0;
                                        (* Entry 'Default': '<S125>:4' *)
                                        (* '<S125>:4:2' FL_sST_MaxChargeCurrent = MaxChargeCurrentBatt *)
                                        FL_sST_MaxChargeCurrent := MaxChargeCurrentBatt;
                                        (* '<S125>:4:3' REQ_HV_Open_Batt1 = false *)
                                        REQ_HV_Open_Batt1 := FALSE;
                                        (* '<S125>:4:4' REQ_HV_Open_Batt2 = false *)
                                        REQ_HV_Open_Batt2 := FALSE;
                                        (* '<S125>:4:5' REQ_HV_Open_Batt3 = false *)
                                        REQ_HV_Open_Batt3 := FALSE;
                                        (* '<S125>:4:6' BatteryReadyToShutDown = true *)
                                        BatteryReadyToShutDown := TRUE;
                                    ELSE 
                                        (* '<S125>:6:2' FL_sST_MaxChargeCurrent = (FL_sST_MaxChargeCurrent - CurrentReductionConstant) *)
                                        FL_sST_MaxChargeCurrent := FL_sST_MaxChargeCurrent - CurrentReductionConstant;
                                        (* '<S125>:6:3' REQ_HV_Open_Batt1 = false *)
                                        REQ_HV_Open_Batt1 := FALSE;
                                        (* '<S125>:6:4' REQ_HV_Open_Batt2 = false *)
                                        REQ_HV_Open_Batt2 := FALSE;
                                        (* '<S125>:6:5' REQ_HV_Open_Batt3 = false *)
                                        REQ_HV_Open_Batt3 := FALSE;
                                        (* '<S125>:6:6' BatteryReadyToShutDown = false *)
                                        BatteryReadyToShutDown := FALSE;
                                    END_IF;

                                END_IF;

                            END_IF;

                        END_IF;

                    END_IF;

                ELSE
                    (* During 'Stop': '<S125>:29' *)
                    (* '<S125>:29:2' FL_sST_MaxChargeCurrent = 0; *)
                    FL_sST_MaxChargeCurrent := 0.0;
                    (* '<S125>:29:3' BatteryReadyToShutDown = true *)
                    BatteryReadyToShutDown := TRUE;
            END_CASE;

        END_IF;

        (* End of Chart: '<S110>/BattChargeFcn' *)
END_CASE;

END_FUNCTION_BLOCK

// Device/Application/Chart_REQ_MAIN_MINUS
FUNCTION_BLOCK Chart_REQ_MAIN_MINUS
VAR_INPUT
	ssMethodType: SINT;
	In: BOOL;
	CM_SafeToSD: BOOL;
	KL15_CM_disable: BOOL;
	System_ESD: BOOL;
	System_SD: BOOL;
	b_Reset: BOOL;
END_VAR
VAR_OUTPUT
	REQ_MainHV_ON_MINUS: BOOL;
END_VAR
VAR
	temporalCounter_i1: PLC_CODER_TIMER;
	is_c20_ChiefMaster: USINT;
	is_active_c20_ChiefMaster: USINT;
	temp1: BOOL;
END_VAR



CASE ssMethodType OF
    SS_INITIALIZE: 
        temporalCounter_i1(timerAction := 1, maxTime := 0);
        is_active_c20_ChiefMaster := 0;
        is_c20_ChiefMaster := ChiefMaster_IN_NO_ACTIVE_CHILD_h;
        REQ_MainHV_ON_MINUS := FALSE;
    SS_OUTPUT: 
        (* Chart: '<S13>/Chart_REQ_MAIN_MINUS' *)
        (* Gateway: ChiefMaster/Flow Logic/BDU Control/BDUSystem/Chart_REQ_MAIN_MINUS *)
        (* During: ChiefMaster/Flow Logic/BDU Control/BDUSystem/Chart_REQ_MAIN_MINUS *)

        IF is_active_c20_ChiefMaster = 0 THEN 
            (* Entry: ChiefMaster/Flow Logic/BDU Control/BDUSystem/Chart_REQ_MAIN_MINUS *)
            is_active_c20_ChiefMaster := 1;
            (* Entry Internal: ChiefMaster/Flow Logic/BDU Control/BDUSystem/Chart_REQ_MAIN_MINUS *)
            (* Transition: '<S16>:4' *)
            is_c20_ChiefMaster := ChiefMaster_IN_Default_a;
            temporalCounter_i1(timerAction := 1, maxTime := 0);
            (* Entry 'Default': '<S16>:3' *)
            (* '<S16>:3:2' REQ_MainHV_ON_MINUS = false *)
            REQ_MainHV_ON_MINUS := FALSE;
        ELSE 
            temp1 := FALSE;

            CASE is_c20_ChiefMaster OF
                ChiefMaster_IN_Default_a: 
                    (* During 'Default': '<S16>:3' *)
                    (* '<S16>:7:1' sf_internal_predicateOutput = after(5,sec) &&... *)
                    (* '<S16>:7:2' System_ESD == false &&... *)
                    (* '<S16>:7:3' System_SD == false &&... *)
                    (* '<S16>:7:4' KL15_CM_disable == false &&... *)
                    (* '<S16>:7:5' Reset == false &&... *)
                    (* '<S16>:7:6' In == true; *)
                    temporalCounter_i1(timerAction := 2, maxTime := 5000);

                    IF temporalCounter_i1.done THEN 

                        IF (((( NOT System_ESD) AND ( NOT System_SD)) AND ( NOT KL15_CM_disable)) AND ( NOT b_Reset)) AND In THEN 
                            (* Transition: '<S16>:7' *)
                            is_c20_ChiefMaster := ChiefMaster_IN_RELMinusClose;
                            (* Entry 'RELMinusClose': '<S16>:6' *)
                            (* '<S16>:6:2' REQ_MainHV_ON_MINUS = true *)
                            REQ_MainHV_ON_MINUS := TRUE;
                        ELSE 
                            (* '<S16>:3:2' REQ_MainHV_ON_MINUS = false *)
                            REQ_MainHV_ON_MINUS := FALSE;
                        END_IF;

                    ELSE 
                        (* '<S16>:3:2' REQ_MainHV_ON_MINUS = false *)
                        REQ_MainHV_ON_MINUS := FALSE;
                    END_IF;

                ChiefMaster_IN_Hold: 
                    (* During 'Hold': '<S16>:14' *)
                    (* '<S16>:15:1' sf_internal_predicateOutput = CM_SafeToSD == true; *)

                    IF CM_SafeToSD THEN 
                        (* Transition: '<S16>:15' *)
                        temp1 := TRUE;
                    ELSE 
                        (* '<S16>:37:1' sf_internal_predicateOutput = after(5,sec); *)
                        temporalCounter_i1(timerAction := 2, maxTime := 5000);

                        IF temporalCounter_i1.done AND System_ESD THEN 
                            (* Transition: '<S16>:37' *)
                            (* '<S16>:38:1' sf_internal_predicateOutput = System_ESD == true; *)
                            (* Transition: '<S16>:38' *)
                            temp1 := TRUE;
                        END_IF;

                    END_IF;

                ELSE
                    (* During 'RELMinusClose': '<S16>:6' *)
                    (* '<S16>:11:1' sf_internal_predicateOutput = System_SD == true ||... *)
                    (* '<S16>:11:2' KL15_CM_disable == true ||... *)
                    (* '<S16>:11:3' Reset == true; *)

                    IF (System_SD OR KL15_CM_disable) OR b_Reset THEN 
                        (* Transition: '<S16>:11' *)
                        is_c20_ChiefMaster := ChiefMaster_IN_Hold;
                        temporalCounter_i1(timerAction := 1, maxTime := 0);
                        (* Entry 'Hold': '<S16>:14' *)
                    ELSE 
                        (* '<S16>:6:2' REQ_MainHV_ON_MINUS = true *)
                        REQ_MainHV_ON_MINUS := TRUE;
                    END_IF;

            END_CASE;


            IF temp1 THEN 
                is_c20_ChiefMaster := ChiefMaster_IN_Default_a;
                temporalCounter_i1(timerAction := 1, maxTime := 0);
                (* Entry 'Default': '<S16>:3' *)
                (* '<S16>:3:2' REQ_MainHV_ON_MINUS = false *)
                REQ_MainHV_ON_MINUS := FALSE;
            END_IF;

        END_IF;

        (* End of Chart: '<S13>/Chart_REQ_MAIN_MINUS' *)
END_CASE;

END_FUNCTION_BLOCK

// Device/Application/Chart_WeldingDetection
FUNCTION_BLOCK Chart_WeldingDetection
VAR_INPUT
	ssMethodType: SINT;
	LoadVtg: REAL;
	SystemVtg: REAL;
	In: BOOL;
END_VAR
VAR_OUTPUT
	MainHV_Minus_Welded: BOOL;
	MainHV_Plus_Welded: BOOL;
	REQ_MainHV_ON_MINUS: BOOL;
	REQ_MainHV_ON_PLUS: BOOL;
	WeldingDetection_Status: USINT;
END_VAR
VAR
	is_c47_ChiefMaster: USINT;
	temporalCounter_i1: PLC_CODER_TIMER;
	is_active_c47_ChiefMaster: USINT;
END_VAR



CASE ssMethodType OF
    SS_INITIALIZE: 
        temporalCounter_i1(timerAction := 1, maxTime := 0);
        is_active_c47_ChiefMaster := 0;
        is_c47_ChiefMaster := ChiefMaster_IN_NO_ACTIVE_CHILD_e;
        MainHV_Minus_Welded := FALSE;
        MainHV_Plus_Welded := FALSE;
        REQ_MainHV_ON_MINUS := FALSE;
        REQ_MainHV_ON_PLUS := FALSE;
        WeldingDetection_Status := 0;
    SS_OUTPUT: 
        (* Chart: '<S22>/Chart_WeldingDetection' *)
        (* Gateway: ChiefMaster/Flow Logic/BDU Control/BDUSystem/Subsystem2/Chart_WeldingDetection *)
        (* During: ChiefMaster/Flow Logic/BDU Control/BDUSystem/Subsystem2/Chart_WeldingDetection *)

        IF is_active_c47_ChiefMaster = 0 THEN 
            (* Entry: ChiefMaster/Flow Logic/BDU Control/BDUSystem/Subsystem2/Chart_WeldingDetection *)
            is_active_c47_ChiefMaster := 1;
            (* Entry Internal: ChiefMaster/Flow Logic/BDU Control/BDUSystem/Subsystem2/Chart_WeldingDetection *)
            (* Transition: '<S30>:2' *)
            is_c47_ChiefMaster := ChiefMaster_IN_Default_b;
            (* Entry 'Default': '<S30>:1' *)
            (* '<S30>:1:2' REQ_MainHV_ON_PLUS = false *)
            REQ_MainHV_ON_PLUS := FALSE;
            (* '<S30>:1:3' REQ_MainHV_ON_MINUS = false *)
            REQ_MainHV_ON_MINUS := FALSE;
            (* '<S30>:1:4' MainHV_Minus_Welded = false *)
            MainHV_Minus_Welded := FALSE;
            (* '<S30>:1:5' MainHV_Plus_Welded = false *)
            MainHV_Plus_Welded := FALSE;
            (* '<S30>:1:6' WeldingDetection_Status = uint8(0); *)
            WeldingDetection_Status := 0;
        ELSE 

            CASE is_c47_ChiefMaster OF
                ChiefMaster_IN_Default_b: 
                    (* During 'Default': '<S30>:1' *)
                    (* '<S30>:41:1' sf_internal_predicateOutput = In == true; *)

                    IF In THEN 
                        (* Transition: '<S30>:41' *)
                        is_c47_ChiefMaster := b_ChiefMaster_IN_Open;
                        temporalCounter_i1(timerAction := 1, maxTime := 0);
                        (* Entry 'Open': '<S30>:40' *)
                        (* '<S30>:40:2' REQ_MainHV_ON_PLUS = false *)
                        REQ_MainHV_ON_PLUS := FALSE;
                        (* '<S30>:40:3' REQ_MainHV_ON_MINUS = false *)
                        REQ_MainHV_ON_MINUS := FALSE;
                        (* '<S30>:40:4' MainHV_Minus_Welded = false *)
                        MainHV_Minus_Welded := FALSE;
                        (* '<S30>:40:5' MainHV_Plus_Welded = false *)
                        MainHV_Plus_Welded := FALSE;
                    ELSE 
                        (* '<S30>:1:2' REQ_MainHV_ON_PLUS = false *)
                        REQ_MainHV_ON_PLUS := FALSE;
                        (* '<S30>:1:3' REQ_MainHV_ON_MINUS = false *)
                        REQ_MainHV_ON_MINUS := FALSE;
                        (* '<S30>:1:4' MainHV_Minus_Welded = false *)
                        MainHV_Minus_Welded := FALSE;
                        (* '<S30>:1:5' MainHV_Plus_Welded = false *)
                        MainHV_Plus_Welded := FALSE;
                        (* '<S30>:1:6' WeldingDetection_Status = uint8(0); *)
                        WeldingDetection_Status := 0;
                    END_IF;

                ChiefMaster_IN_Default3: 
                    (* During 'Default3': '<S30>:16' *)
                    (* '<S30>:25:1' sf_internal_predicateOutput = after(5,sec); *)
                    temporalCounter_i1(timerAction := 2, maxTime := 5000);

                    IF temporalCounter_i1.done THEN 
                        (* Transition: '<S30>:25' *)
                        is_c47_ChiefMaster := ChiefMaster_IN_ErrorPlus;
                        (* Entry 'ErrorPlus': '<S30>:24' *)
                        (* '<S30>:24:2' MainHV_Plus_Welded = true *)
                        MainHV_Plus_Welded := TRUE;
                        (* '<S30>:24:3' WeldingDetection_Status = uint8(2); *)
                        WeldingDetection_Status := 2;
                    ELSE 
                        (* '<S30>:29:1' sf_internal_predicateOutput = LoadVtg <= 20; *)

                        IF LoadVtg <= 20.0 THEN 
                            (* Transition: '<S30>:29' *)
                            is_c47_ChiefMaster := ChiefMaster_IN_Open1;
                            (* Entry 'Open1': '<S30>:28' *)
                            (* '<S30>:28:2' REQ_MainHV_ON_PLUS = false *)
                            REQ_MainHV_ON_PLUS := FALSE;
                            (* '<S30>:28:3' REQ_MainHV_ON_MINUS = false *)
                            REQ_MainHV_ON_MINUS := FALSE;
                            (* '<S30>:28:4' MainHV_Minus_Welded = false *)
                            MainHV_Minus_Welded := FALSE;
                            (* '<S30>:28:5' MainHV_Plus_Welded = false *)
                            MainHV_Plus_Welded := FALSE;
                            (* '<S30>:28:6' WeldingDetection_Status = uint8(1); *)
                            WeldingDetection_Status := 1;
                        ELSE 
                            (* '<S30>:16:2' REQ_MainHV_ON_PLUS = false *)
                            REQ_MainHV_ON_PLUS := FALSE;
                        END_IF;

                    END_IF;

                ChiefMaster_IN_Error: 
                    (* During 'Error': '<S30>:38' *)
                    (* '<S30>:38:2' MainHV_Minus_Welded = true *)
                    MainHV_Minus_Welded := TRUE;
                    (* '<S30>:38:3' MainHV_Plus_Welded = true *)
                    MainHV_Plus_Welded := TRUE;
                    (* '<S30>:38:4' WeldingDetection_Status = uint8(2); *)
                    WeldingDetection_Status := 2;
                ChiefMaster_IN_ErrorMinus: 
                    (* During 'ErrorMinus': '<S30>:22' *)
                    (* '<S30>:22:2' MainHV_Minus_Welded = true *)
                    MainHV_Minus_Welded := TRUE;
                    (* '<S30>:22:3' WeldingDetection_Status = uint8(2); *)
                    WeldingDetection_Status := 2;
                ChiefMaster_IN_ErrorPlus: 
                    (* During 'ErrorPlus': '<S30>:24' *)
                    (* '<S30>:24:2' MainHV_Plus_Welded = true *)
                    MainHV_Plus_Welded := TRUE;
                    (* '<S30>:24:3' WeldingDetection_Status = uint8(2); *)
                    WeldingDetection_Status := 2;
                ChiefMaster_IN_ErrorVoltage: 
                    (* During 'ErrorVoltage': '<S30>:45' *)
                    (* '<S30>:45:2' WeldingDetection_Status = uint8(2); *)
                    WeldingDetection_Status := 2;
                ChiefMaster_IN_Minus_Close: 
                    (* During 'Minus_Close': '<S30>:12' *)
                    (* '<S30>:17:1' sf_internal_predicateOutput = abs(LoadVtg - SystemVtg) <= 5; *)

                    IF ABS(LoadVtg - SystemVtg) <= 5.0 THEN 
                        (* Transition: '<S30>:17' *)
                        is_c47_ChiefMaster := ChiefMaster_IN_Default3;
                        temporalCounter_i1(timerAction := 1, maxTime := 0);
                        (* Entry 'Default3': '<S30>:16' *)
                        (* '<S30>:16:2' REQ_MainHV_ON_PLUS = false *)
                        REQ_MainHV_ON_PLUS := FALSE;
                    ELSE 
                        (* '<S30>:46:1' sf_internal_predicateOutput = after(5,sec); *)
                        temporalCounter_i1(timerAction := 2, maxTime := 5000);

                        IF temporalCounter_i1.done THEN 
                            (* Transition: '<S30>:46' *)
                            is_c47_ChiefMaster := ChiefMaster_IN_ErrorVoltage;
                            (* Entry 'ErrorVoltage': '<S30>:45' *)
                            (* '<S30>:45:2' WeldingDetection_Status = uint8(2); *)
                            WeldingDetection_Status := 2;
                        ELSE 
                            (* '<S30>:12:2' REQ_MainHV_ON_MINUS = true *)
                            REQ_MainHV_ON_MINUS := TRUE;
                        END_IF;

                    END_IF;

                b_ChiefMaster_IN_Open: 
                    (* During 'Open': '<S30>:40' *)
                    (* '<S30>:5:1' sf_internal_predicateOutput = LoadVtg <= 20; *)

                    IF LoadVtg <= 20.0 THEN 
                        (* Transition: '<S30>:5' *)
                        is_c47_ChiefMaster := ChiefMaster_IN_Plus_Close;
                        temporalCounter_i1(timerAction := 1, maxTime := 0);
                        (* Entry 'Plus_Close': '<S30>:4' *)
                        (* '<S30>:4:2' REQ_MainHV_ON_PLUS = true *)
                        REQ_MainHV_ON_PLUS := TRUE;
                    ELSE 
                        (* '<S30>:42:1' sf_internal_predicateOutput = after(5,sec); *)
                        temporalCounter_i1(timerAction := 2, maxTime := 5000);

